Yaskawa INFORM job: vendrediTRJ4.JBI

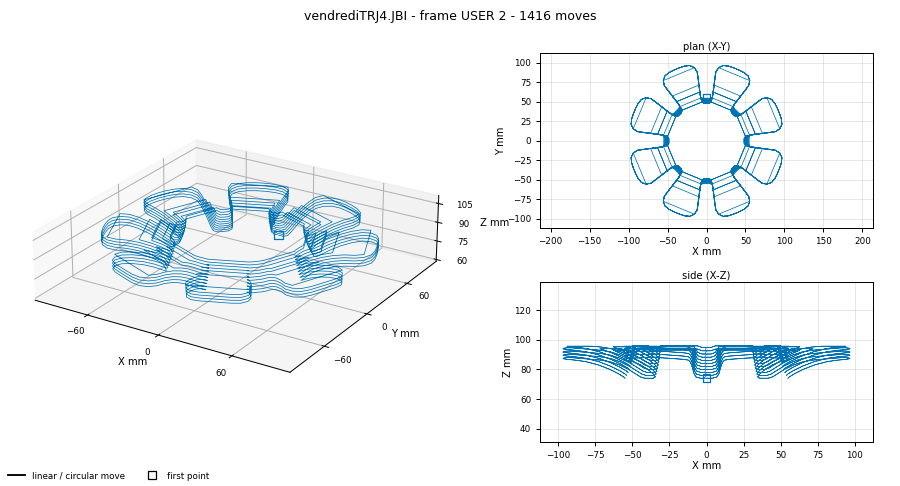
[picture p0: tool path of vendrediTRJ4.JBI in frame USER 2, 1416 of 1416 moves have a stored position in this frame; points joined in program order, loops and branches not executed]
/JOB
//NAME vendrediTRJ4
///FOLDERNAME DEMO
//POS
///NPOS 1416,0,1416,0,0,0
///USER 2
///TOOL 7
///POSTYPE USER
///RECTAN
///RCONF 1,0,0,0,0,0,0,0,0,0,0,0,0,0,0,0,0,0,0,0,0,0,0,0
C00000=0.000,54.840,74.049,-180.0000,29.7413,-14490.0000
C00001=1.666,54.823,74.024,-179.8067,29.7500,-14491.7406
C00002=4.048,54.790,74.062,173.8586,28.2915,-14494.2255
C00003=7.088,55.804,74.943,167.0788,9.5543,-14497.2387
C00004=8.393,59.388,77.145,-177.8370,-0.0706,-14498.0440
C00005=9.180,65.335,80.122,-176.4294,-0.0310,-14497.9981
C00006=10.089,72.980,83.074,-176.0907,-0.0153,-14497.8709
C00007=11.094,81.206,85.240,-175.9759,-0.0117,-14497.7793
C00008=12.226,88.613,86.276,-176.2817,-0.6456,-14497.8555
C00009=15.808,94.009,86.813,-178.2035,-1.5233,-14499.5452
C00010=21.475,96.642,87.246,-179.5823,-1.0342,-14502.5282
C00011=28.048,95.980,87.679,179.9973,-0.0724,-14506.2898
C00012=34.856,93.728,87.962,179.9966,-0.0074,-14510.3994
C00013=41.629,90.922,87.962,179.9972,-0.0076,-14514.6009
C00014=48.035,87.701,87.679,-179.9999,-0.0718,-14518.7101
C00015=53.151,83.521,87.246,179.5838,-1.0323,-14522.4718
C00016=55.296,77.652,86.813,178.2066,-1.5235,-14525.4547
C00017=54.014,71.304,86.276,176.2804,-0.6460,-14527.1446
C00018=49.577,65.266,85.240,175.9790,-0.0155,-14527.2208
C00019=44.470,58.738,83.074,176.0895,-0.0120,-14527.1290
C00020=39.708,52.690,80.122,176.4261,-0.0301,-14527.0022
C00021=36.059,47.928,77.145,177.8373,-0.0709,-14526.9563
C00022=34.447,44.472,74.943,-167.0757,9.5522,-14527.7605
C00023=35.880,41.605,74.062,-173.8568,28.2919,-14530.7744
C00024=37.588,39.944,74.024,179.8046,29.7498,-14533.2595
C00025=38.778,38.778,74.049,-180.0000,29.7416,-14535.0000
C00026=39.943,37.588,74.024,-179.8042,29.7498,-14536.7398
C00027=41.605,35.880,74.062,173.8533,28.2853,-14539.2256
C00028=44.472,34.447,74.943,167.0757,9.5522,-14542.2395
C00029=47.928,36.059,77.145,-177.8373,-0.0709,-14543.0437
C00030=52.690,39.708,80.122,-176.4261,-0.0301,-14542.9978
C00031=58.738,44.470,83.074,-176.0895,-0.0120,-14542.8710
C00032=65.266,49.577,85.240,-175.9790,-0.0155,-14542.7792
C00033=71.304,54.014,86.276,-176.2804,-0.6460,-14542.8554
C00034=77.652,55.296,86.813,-178.2066,-1.5235,-14544.5453
C00035=83.521,53.151,87.246,-179.5838,-1.0323,-14547.5282
C00036=87.701,48.035,87.679,179.9999,-0.0718,-14551.2899
C00037=90.922,41.629,87.962,-179.9972,-0.0076,-14555.3991
C00038=93.728,34.856,87.962,-179.9966,-0.0074,-14559.6006
C00039=95.980,28.048,87.679,-179.9973,-0.0724,-14563.7102
C00040=96.642,21.475,87.246,179.5823,-1.0342,-14567.4718
C00041=94.009,15.808,86.813,178.2035,-1.5233,-14570.4548
C00042=88.613,12.226,86.276,176.2817,-0.6456,-14572.1445
C00043=81.206,11.094,85.240,175.9759,-0.0117,-14572.2207
C00044=72.980,10.089,83.074,176.0907,-0.0153,-14572.1291
C00045=65.335,9.180,80.122,176.4294,-0.0310,-14572.0019
C00046=59.388,8.393,77.145,177.8370,-0.0706,-14571.9560
C00047=55.804,7.088,74.943,-167.0788,9.5543,-14572.7613
C00048=54.790,4.048,74.062,-173.8586,28.2915,-14575.7745
C00049=54.823,1.666,74.024,179.8067,29.7500,-14578.2594
C00050=54.840,0.000,74.049,180.0000,29.7413,-14580.0000
C00051=54.823,-1.665,74.024,-179.8061,29.7500,-14581.7396
C00052=54.790,-4.048,74.062,173.8593,28.2888,-14584.2255
C00053=55.804,-7.088,74.943,167.0788,9.5543,-14587.2387
C00054=59.388,-8.393,77.145,-177.8370,-0.0706,-14588.0440
C00055=65.335,-9.180,80.122,-176.4294,-0.0310,-14587.9981
C00056=72.980,-10.089,83.074,-176.0907,-0.0153,-14587.8709
C00057=81.206,-11.094,85.240,-175.9759,-0.0117,-14587.7793
C00058=88.613,-12.226,86.276,-176.2817,-0.6456,-14587.8555
C00059=94.009,-15.808,86.813,-178.2035,-1.5233,-14589.5452
C00060=96.642,-21.475,87.246,-179.5823,-1.0342,-14592.5282
C00061=95.980,-28.048,87.679,179.9973,-0.0724,-14596.2898
C00062=93.728,-34.856,87.962,179.9966,-0.0074,-14600.3994
C00063=90.922,-41.629,87.962,179.9972,-0.0076,-14604.6009
C00064=87.701,-48.035,87.679,-179.9999,-0.0718,-14608.7101
C00065=83.521,-53.151,87.246,179.5838,-1.0323,-14612.4718
C00066=77.652,-55.296,86.813,178.2066,-1.5235,-14615.4547
C00067=71.304,-54.014,86.276,176.2804,-0.6460,-14617.1446
C00068=65.266,-49.577,85.240,175.9790,-0.0155,-14617.2208
C00069=58.738,-44.470,83.074,176.0895,-0.0120,-14617.1290
C00070=52.690,-39.708,80.122,176.4261,-0.0301,-14617.0022
C00071=47.928,-36.059,77.145,177.8373,-0.0709,-14616.9563
C00072=44.472,-34.447,74.943,-167.0757,9.5522,-14617.7605
C00073=41.605,-35.880,74.062,-173.8568,28.2919,-14620.7744
C00074=39.944,-37.588,74.024,179.8046,29.7498,-14623.2595
C00075=38.778,-38.778,74.049,180.0000,29.7416,-14625.0000
C00076=37.588,-39.943,74.024,-179.8042,29.7498,-14626.7398
C00077=35.880,-41.605,74.062,173.8533,28.2853,-14629.2256
C00078=34.447,-44.472,74.943,167.0757,9.5522,-14632.2395
C00079=36.059,-47.928,77.145,-177.8373,-0.0709,-14633.0437
C00080=39.708,-52.690,80.122,-176.4261,-0.0301,-14632.9978
C00081=44.470,-58.738,83.074,-176.0895,-0.0120,-14632.8710
C00082=49.577,-65.266,85.240,-175.9790,-0.0155,-14632.7792
C00083=54.014,-71.304,86.276,-176.2804,-0.6460,-14632.8554
C00084=55.296,-77.652,86.813,-178.2066,-1.5235,-14634.5453
C00085=53.151,-83.521,87.246,-179.5838,-1.0323,-14637.5282
C00086=48.035,-87.701,87.679,179.9999,-0.0718,-14641.2899
C00087=41.629,-90.922,87.962,-179.9972,-0.0076,-14645.3991
C00088=34.856,-93.728,87.962,-179.9966,-0.0074,-14649.6006
C00089=28.048,-95.980,87.679,-179.9973,-0.0724,-14653.7102
C00090=21.475,-96.642,87.246,179.5823,-1.0342,-14657.4718
C00091=15.808,-94.009,86.813,178.2035,-1.5233,-14660.4548
C00092=12.226,-88.613,86.276,176.2817,-0.6456,-14662.1445
C00093=11.094,-81.206,85.240,175.9759,-0.0117,-14662.2207
C00094=10.089,-72.980,83.074,176.0907,-0.0153,-14662.1291
C00095=9.180,-65.335,80.122,176.4294,-0.0310,-14662.0019
C00096=8.393,-59.388,77.145,177.8370,-0.0706,-14661.9560
C00097=7.088,-55.804,74.943,-167.0788,9.5543,-14662.7613
C00098=4.048,-54.790,74.062,-173.8586,28.2915,-14665.7745
C00099=1.666,-54.823,74.024,179.8067,29.7500,-14668.2594
C00100=0.000,-54.840,74.049,-180.0000,29.7413,-14670.0000
C00101=-1.665,-54.823,74.024,-179.8061,29.7500,-14671.7396
C00102=-4.048,-54.790,74.062,173.8593,28.2888,-14674.2255
C00103=-7.088,-55.804,74.943,167.0788,9.5543,-14677.2387
C00104=-8.393,-59.388,77.145,-177.8370,-0.0706,-14678.0440
C00105=-9.180,-65.335,80.122,-176.4294,-0.0310,-14677.9981
C00106=-10.089,-72.980,83.074,-176.0907,-0.0153,-14677.8709
C00107=-11.094,-81.206,85.240,-175.9759,-0.0117,-14677.7793
C00108=-12.226,-88.613,86.276,-176.2817,-0.6456,-14677.8555
C00109=-15.808,-94.009,86.813,-178.2035,-1.5233,-14679.5452
C00110=-21.475,-96.642,87.246,-179.5823,-1.0342,-14682.5282
C00111=-28.048,-95.980,87.679,179.9973,-0.0724,-14686.2898
C00112=-34.856,-93.728,87.962,179.9966,-0.0074,-14690.3994
C00113=-41.629,-90.922,87.962,179.9972,-0.0076,-14694.6009
C00114=-48.035,-87.701,87.679,-179.9999,-0.0718,-14698.7101
C00115=-53.151,-83.521,87.246,179.5838,-1.0323,-14702.4718
C00116=-55.296,-77.652,86.813,178.2066,-1.5235,-14705.4547
C00117=-54.014,-71.304,86.276,176.2804,-0.6460,-14707.1446
C00118=-49.577,-65.266,85.240,175.9790,-0.0155,-14707.2208
C00119=-44.470,-58.738,83.074,176.0895,-0.0120,-14707.1290
C00120=-39.708,-52.690,80.122,176.4261,-0.0301,-14707.0022
C00121=-36.059,-47.928,77.145,177.8373,-0.0709,-14706.9563
C00122=-34.447,-44.472,74.943,-167.0757,9.5522,-14707.7605
C00123=-35.880,-41.605,74.062,-173.8568,28.2919,-14710.7744
C00124=-37.588,-39.944,74.024,179.8046,29.7498,-14713.2595
C00125=-38.778,-38.778,74.049,-180.0000,29.7416,-14715.0000
C00126=-39.943,-37.588,74.024,-179.8042,29.7498,-14716.7398
C00127=-41.605,-35.880,74.062,173.8533,28.2853,-14719.2256
C00128=-44.472,-34.447,74.943,167.0757,9.5522,-14722.2395
C00129=-47.928,-36.059,77.145,-177.8373,-0.0709,-14723.0437
C00130=-52.690,-39.708,80.122,-176.4261,-0.0301,-14722.9978
C00131=-58.738,-44.470,83.074,-176.0895,-0.0120,-14722.8710
C00132=-65.266,-49.577,85.240,-175.9790,-0.0155,-14722.7792
C00133=-71.304,-54.014,86.276,-176.2804,-0.6460,-14722.8554
C00134=-77.652,-55.296,86.813,-178.2066,-1.5235,-14724.5453
C00135=-83.521,-53.151,87.246,-179.5838,-1.0323,-14727.5282
C00136=-87.701,-48.035,87.679,179.9999,-0.0718,-14731.2899
C00137=-90.922,-41.629,87.962,-179.9972,-0.0076,-14735.3991
C00138=-93.728,-34.856,87.962,-179.9966,-0.0074,-14739.6006
C00139=-95.980,-28.048,87.679,-179.9973,-0.0724,-14743.7102
C00140=-96.642,-21.475,87.246,179.5823,-1.0342,-14747.4718
C00141=-94.009,-15.808,86.813,178.2035,-1.5233,-14750.4548
C00142=-88.613,-12.226,86.276,176.2817,-0.6456,-14752.1445
C00143=-81.206,-11.094,85.240,175.9759,-0.0117,-14752.2207
C00144=-72.980,-10.089,83.074,176.0907,-0.0153,-14752.1291
C00145=-65.335,-9.180,80.122,176.4294,-0.0310,-14752.0019
C00146=-59.388,-8.393,77.145,177.8370,-0.0706,-14751.9560
C00147=-55.804,-7.088,74.943,-167.0788,9.5543,-14752.7613
C00148=-54.790,-4.048,74.062,-173.8586,28.2915,-14755.7745
C00149=-54.823,-1.666,74.024,179.8067,29.7500,-14758.2594
C00150=-54.840,0.000,74.049,-180.0000,29.7413,-14760.0000
C00151=-54.823,1.665,74.024,-179.8061,29.7500,-14761.7396
C00152=-54.790,4.048,74.062,173.8593,28.2888,-14764.2255
C00153=-55.804,7.088,74.943,167.0788,9.5543,-14767.2387
C00154=-59.388,8.393,77.145,-177.8370,-0.0706,-14768.0440
C00155=-65.335,9.180,80.122,-176.4294,-0.0310,-14767.9981
C00156=-72.980,10.089,83.074,-176.0907,-0.0153,-14767.8709
C00157=-81.206,11.094,85.240,-175.9759,-0.0117,-14767.7793
C00158=-88.613,12.226,86.276,-176.2817,-0.6456,-14767.8555
C00159=-94.009,15.808,86.813,-178.2035,-1.5233,-14769.5452
C00160=-96.642,21.475,87.246,-179.5823,-1.0342,-14772.5282
C00161=-95.980,28.048,87.679,179.9973,-0.0724,-14776.2898
C00162=-93.728,34.856,87.962,179.9966,-0.0074,-14780.3994
C00163=-90.922,41.629,87.962,179.9972,-0.0076,-14784.6009
C00164=-87.701,48.035,87.679,-179.9999,-0.0718,-14788.7101
C00165=-83.521,53.151,87.246,179.5838,-1.0323,-14792.4718
C00166=-77.652,55.296,86.813,178.2066,-1.5235,-14795.4547
C00167=-71.304,54.014,86.276,176.2804,-0.6460,-14797.1446
C00168=-65.266,49.577,85.240,175.9790,-0.0155,-14797.2208
C00169=-58.738,44.470,83.074,176.0895,-0.0120,-14797.1290
C00170=-52.690,39.708,80.122,176.4261,-0.0301,-14797.0022
C00171=-47.928,36.059,77.145,177.8373,-0.0709,-14796.9563
C00172=-44.472,34.447,74.943,-167.0757,9.5522,-14797.7605
C00173=-41.605,35.880,74.062,-173.8568,28.2919,-14800.7744
C00174=-39.944,37.588,74.024,179.8046,29.7498,-14803.2595
C00175=-38.778,38.778,74.049,-180.0000,29.7416,-14805.0000
C00176=-37.588,39.943,74.024,-179.8042,29.7498,-14806.7398
C00177=-35.880,41.605,74.062,173.8533,28.2853,-14809.2256
C00178=-34.447,44.472,74.943,167.0757,9.5522,-14812.2395
C00179=-36.059,47.928,77.145,-177.8373,-0.0709,-14813.0437
C00180=-39.708,52.690,80.122,-176.4261,-0.0301,-14812.9978
C00181=-44.470,58.738,83.074,-176.0895,-0.0120,-14812.8710
C00182=-49.577,65.266,85.240,-175.9790,-0.0155,-14812.7792
C00183=-54.014,71.304,86.276,-176.2804,-0.6460,-14812.8554
C00184=-55.296,77.652,86.813,-178.2066,-1.5235,-14814.5453
C00185=-53.151,83.521,87.246,-179.5838,-1.0323,-14817.5282
C00186=-48.035,87.701,87.679,179.9999,-0.0718,-14821.2899
C00187=-41.629,90.922,87.962,-179.9972,-0.0076,-14825.3991
C00188=-34.856,93.728,87.962,-179.9966,-0.0074,-14829.6006
C00189=-28.048,95.980,87.679,-179.9973,-0.0724,-14833.7102
C00190=-21.475,96.642,87.246,179.5823,-1.0342,-14837.4718
C00191=-15.808,94.009,86.813,178.2035,-1.5233,-14840.4548
C00192=-12.226,88.613,86.276,176.2817,-0.6456,-14842.1445
C00193=-11.094,81.206,85.240,175.9759,-0.0117,-14842.2207
C00194=-10.089,72.980,83.074,176.0907,-0.0153,-14842.1291
C00195=-9.180,65.335,80.122,176.4294,-0.0310,-14842.0019
C00196=-8.393,59.388,77.145,177.8370,-0.0706,-14841.9560
C00197=-7.088,55.804,74.943,-167.0788,9.5543,-14842.7613
C00198=-4.048,54.790,74.062,-173.8593,28.2888,-14845.7745
C00199=-1.665,54.823,74.024,179.8061,29.7500,-14848.2604
C00200=0.000,53.776,75.975,180.0000,28.1001,-14850.0000
C00201=1.568,53.762,75.948,-179.8334,28.1117,-14851.6706
C00202=3.884,53.739,75.988,174.0567,26.6026,-14854.1339
C00203=6.894,54.818,76.900,168.1623,8.4382,-14857.1680
C00204=8.175,58.565,79.173,-177.8225,-0.0548,-14857.9465
C00205=8.965,64.737,82.228,-176.7507,-0.0188,-14857.8844
C00206=9.898,72.606,85.234,-176.6314,-0.0094,-14857.7630
C00207=10.924,81.005,87.424,-176.6961,-0.0057,-14857.6803
C00208=12.061,88.524,88.468,-177.0328,-0.5045,-14857.7585
C00209=15.662,93.991,89.008,-178.5867,-1.1939,-14859.4604
C00210=21.365,96.662,89.443,-179.6771,-0.7971,-14862.4636
C00211=27.983,96.002,89.878,179.9979,-0.0543,-14866.2505
C00212=34.834,93.736,90.162,-179.9980,-0.0054,-14870.3860
C00213=41.650,90.913,90.162,-179.9976,-0.0052,-14874.6140
C00214=48.097,87.670,89.878,179.9969,-0.0540,-14878.7498
C00215=53.243,83.458,89.443,179.6739,-0.7993,-14882.5363
C00216=55.387,77.537,89.008,178.5849,-1.1940,-14885.5394
C00217=54.067,71.124,88.468,177.0304,-0.5081,-14887.2413
C00218=49.554,65.004,87.424,176.6978,-0.0087,-14887.3191
C00219=44.341,58.339,85.234,176.6315,-0.0113,-14887.2369
C00220=39.437,52.115,82.228,176.7520,-0.0208,-14887.1159
C00221=35.631,47.192,79.173,177.8236,-0.0563,-14887.0536
C00222=33.888,43.637,76.900,-168.1624,8.4405,-14887.8325
C00223=35.253,40.746,75.988,-174.0559,26.5997,-14890.8660
C00224=36.906,39.124,75.948,179.8313,28.1098,-14893.3290
C00225=38.025,38.025,75.975,-180.0000,28.0967,-14895.0000
C00226=39.124,36.906,75.948,-179.8313,28.1098,-14896.6710
C00227=40.746,35.253,75.988,174.0559,26.5997,-14899.1340
C00228=43.637,33.888,76.901,168.1624,8.4405,-14902.1675
C00229=47.192,35.631,79.173,-177.8236,-0.0563,-14902.9464
C00230=52.115,39.437,82.228,-176.7520,-0.0208,-14902.8841
C00231=58.339,44.341,85.234,-176.6315,-0.0113,-14902.7631
C00232=65.004,49.554,87.424,-176.6978,-0.0087,-14902.6809
C00233=71.124,54.067,88.468,-177.0304,-0.5081,-14902.7587
C00234=77.537,55.387,89.008,-178.5849,-1.1940,-14904.4606
C00235=83.458,53.243,89.443,-179.6739,-0.7993,-14907.4637
C00236=87.670,48.097,89.878,-179.9969,-0.0540,-14911.2502
C00237=90.913,41.650,90.162,179.9976,-0.0052,-14915.3860
C00238=93.736,34.834,90.162,179.9980,-0.0054,-14919.6140
C00239=96.002,27.983,89.878,-179.9979,-0.0543,-14923.7495
C00240=96.662,21.365,89.443,179.6771,-0.7971,-14927.5364
C00241=93.991,15.662,89.008,178.5867,-1.1939,-14930.5396
C00242=88.524,12.061,88.468,177.0328,-0.5045,-14932.2415
C00243=81.005,10.924,87.424,176.6961,-0.0057,-14932.3197
C00244=72.606,9.898,85.234,176.6314,-0.0094,-14932.2370
C00245=64.737,8.965,82.228,176.7507,-0.0188,-14932.1156
C00246=58.565,8.175,79.173,177.8225,-0.0548,-14932.0535
C00247=54.818,6.894,76.900,-168.1623,8.4382,-14932.8320
C00248=53.739,3.884,75.988,-174.0567,26.6026,-14935.8661
C00249=53.762,1.568,75.948,179.8334,28.1117,-14938.3294
C00250=53.776,0.000,75.975,180.0000,28.1001,-14940.0000
C00251=53.762,-1.568,75.948,-179.8334,28.1117,-14941.6706
C00252=53.739,-3.885,75.988,174.0562,26.6025,-14944.1349
C00253=54.819,-6.894,76.901,168.1623,8.4383,-14947.1678
C00254=58.565,-8.175,79.173,-177.8225,-0.0548,-14947.9465
C00255=64.737,-8.965,82.228,-176.7507,-0.0188,-14947.8844
C00256=72.606,-9.898,85.234,-176.6314,-0.0094,-14947.7630
C00257=81.005,-10.924,87.424,-176.6961,-0.0057,-14947.6803
C00258=88.524,-12.061,88.468,-177.0328,-0.5045,-14947.7585
C00259=93.991,-15.662,89.008,-178.5867,-1.1939,-14949.4604
C00260=96.662,-21.365,89.443,-179.6771,-0.7971,-14952.4636
C00261=96.002,-27.983,89.878,179.9979,-0.0543,-14956.2505
C00262=93.736,-34.834,90.162,-179.9980,-0.0054,-14960.3860
C00263=90.913,-41.650,90.162,-179.9976,-0.0052,-14964.6140
C00264=87.670,-48.097,89.878,179.9969,-0.0540,-14968.7498
C00265=83.458,-53.243,89.443,179.6739,-0.7993,-14972.5363
C00266=77.537,-55.387,89.008,178.5849,-1.1940,-14975.5394
C00267=71.124,-54.067,88.468,177.0304,-0.5081,-14977.2413
C00268=65.004,-49.554,87.424,176.6978,-0.0087,-14977.3191
C00269=58.339,-44.341,85.234,176.6315,-0.0113,-14977.2369
C00270=52.115,-39.437,82.228,176.7520,-0.0208,-14977.1159
C00271=47.192,-35.631,79.173,177.8236,-0.0563,-14977.0536
C00272=43.637,-33.888,76.900,-168.1624,8.4405,-14977.8325
C00273=40.746,-35.253,75.988,-174.0559,26.5997,-14980.8660
C00274=39.124,-36.906,75.948,179.8313,28.1098,-14983.3290
C00275=38.025,-38.025,75.975,-180.0000,28.0967,-14985.0000
C00276=36.906,-39.124,75.948,-179.8313,28.1098,-14986.6710
C00277=35.253,-40.746,75.988,174.0559,26.5997,-14989.1340
C00278=33.888,-43.637,76.901,168.1624,8.4405,-14992.1675
C00279=35.631,-47.192,79.173,-177.8236,-0.0563,-14992.9464
C00280=39.437,-52.115,82.228,-176.7520,-0.0208,-14992.8841
C00281=44.341,-58.339,85.234,-176.6315,-0.0113,-14992.7631
C00282=49.554,-65.004,87.424,-176.6978,-0.0087,-14992.6809
C00283=54.067,-71.124,88.468,-177.0304,-0.5081,-14992.7587
C00284=55.387,-77.537,89.008,-178.5849,-1.1940,-14994.4606
C00285=53.243,-83.458,89.443,-179.6739,-0.7993,-14997.4637
C00286=48.097,-87.670,89.878,-179.9969,-0.0540,-15001.2502
C00287=41.650,-90.913,90.162,179.9976,-0.0052,-15005.3860
C00288=34.834,-93.736,90.162,179.9980,-0.0054,-15009.6140
C00289=27.983,-96.002,89.878,-179.9979,-0.0543,-15013.7495
C00290=21.365,-96.662,89.443,179.6771,-0.7971,-15017.5364
C00291=15.662,-93.991,89.008,178.5867,-1.1939,-15020.5396
C00292=12.061,-88.524,88.468,177.0328,-0.5045,-15022.2415
C00293=10.924,-81.005,87.424,176.6961,-0.0057,-15022.3197
C00294=9.898,-72.606,85.234,176.6314,-0.0094,-15022.2370
C00295=8.965,-64.737,82.228,176.7507,-0.0188,-15022.1156
C00296=8.175,-58.565,79.173,177.8225,-0.0548,-15022.0535
C00297=6.894,-54.818,76.900,-168.1623,8.4382,-15022.8320
C00298=3.884,-53.739,75.988,-174.0567,26.6026,-15025.8661
C00299=1.568,-53.762,75.948,179.8334,28.1117,-15028.3294
C00300=0.000,-53.776,75.975,180.0000,28.1001,-15030.0000
C00301=-1.568,-53.762,75.948,-179.8334,28.1117,-15031.6706
C00302=-3.885,-53.739,75.988,174.0562,26.6025,-15034.1349
C00303=-6.894,-54.819,76.901,168.1623,8.4383,-15037.1678
C00304=-8.175,-58.565,79.173,-177.8225,-0.0548,-15037.9465
C00305=-8.965,-64.737,82.228,-176.7507,-0.0188,-15037.8844
C00306=-9.898,-72.606,85.234,-176.6314,-0.0094,-15037.7630
C00307=-10.924,-81.005,87.424,-176.6961,-0.0057,-15037.6803
C00308=-12.061,-88.524,88.468,-177.0328,-0.5045,-15037.7585
C00309=-15.662,-93.991,89.008,-178.5867,-1.1939,-15039.4604
C00310=-21.365,-96.662,89.443,-179.6771,-0.7971,-15042.4636
C00311=-27.983,-96.002,89.878,179.9979,-0.0543,-15046.2505
C00312=-34.834,-93.736,90.162,-179.9980,-0.0054,-15050.3860
C00313=-41.650,-90.913,90.162,-179.9976,-0.0052,-15054.6140
C00314=-48.097,-87.670,89.878,179.9969,-0.0540,-15058.7498
C00315=-53.243,-83.458,89.443,179.6739,-0.7993,-15062.5363
C00316=-55.387,-77.537,89.008,178.5849,-1.1940,-15065.5394
C00317=-54.067,-71.124,88.468,177.0304,-0.5081,-15067.2413
C00318=-49.554,-65.004,87.424,176.6978,-0.0087,-15067.3191
C00319=-44.341,-58.339,85.234,176.6315,-0.0113,-15067.2369
C00320=-39.437,-52.115,82.228,176.7520,-0.0208,-15067.1159
C00321=-35.631,-47.192,79.173,177.8236,-0.0563,-15067.0536
C00322=-33.888,-43.637,76.900,-168.1624,8.4405,-15067.8325
C00323=-35.253,-40.746,75.988,-174.0559,26.5997,-15070.8660
C00324=-36.906,-39.124,75.948,179.8313,28.1098,-15073.3290
C00325=-38.025,-38.025,75.975,-180.0000,28.0967,-15075.0000
C00326=-39.124,-36.906,75.948,-179.8313,28.1098,-15076.6710
C00327=-40.746,-35.253,75.988,174.0559,26.5997,-15079.1340
C00328=-43.637,-33.888,76.901,168.1624,8.4405,-15082.1675
C00329=-47.192,-35.631,79.173,-177.8236,-0.0563,-15082.9464
C00330=-52.115,-39.437,82.228,-176.7520,-0.0208,-15082.8841
C00331=-58.339,-44.341,85.234,-176.6315,-0.0113,-15082.7631
C00332=-65.004,-49.554,87.424,-176.6978,-0.0087,-15082.6809
C00333=-71.124,-54.067,88.468,-177.0304,-0.5081,-15082.7587
C00334=-77.537,-55.387,89.008,-178.5849,-1.1940,-15084.4606
C00335=-83.458,-53.243,89.443,-179.6739,-0.7993,-15087.4637
C00336=-87.670,-48.097,89.878,-179.9969,-0.0540,-15091.2502
C00337=-90.913,-41.650,90.162,179.9976,-0.0052,-15095.3860
C00338=-93.736,-34.834,90.162,179.9980,-0.0054,-15099.6140
C00339=-96.002,-27.983,89.878,-179.9979,-0.0543,-15103.7495
C00340=-96.662,-21.365,89.443,179.6771,-0.7971,-15107.5364
C00341=-93.991,-15.662,89.008,178.5867,-1.1939,-15110.5396
C00342=-88.524,-12.061,88.468,177.0328,-0.5045,-15112.2415
C00343=-81.005,-10.924,87.424,176.6961,-0.0057,-15112.3197
C00344=-72.606,-9.898,85.234,176.6314,-0.0094,-15112.2370
C00345=-64.737,-8.965,82.228,176.7507,-0.0188,-15112.1156
C00346=-58.565,-8.175,79.173,177.8225,-0.0548,-15112.0535
C00347=-54.818,-6.894,76.900,-168.1623,8.4382,-15112.8320
C00348=-53.739,-3.884,75.988,-174.0567,26.6026,-15115.8661
C00349=-53.762,-1.568,75.948,179.8334,28.1117,-15118.3294
C00350=-53.776,0.000,75.975,180.0000,28.1001,-15120.0000
C00351=-53.762,1.568,75.948,-179.8334,28.1117,-15121.6706
C00352=-53.739,3.885,75.988,174.0562,26.6025,-15124.1349
C00353=-54.819,6.894,76.901,168.1623,8.4383,-15127.1678
C00354=-58.565,8.175,79.173,-177.8225,-0.0548,-15127.9465
C00355=-64.737,8.965,82.228,-176.7507,-0.0188,-15127.8844
C00356=-72.606,9.898,85.234,-176.6314,-0.0094,-15127.7630
C00357=-81.005,10.924,87.424,-176.6961,-0.0057,-15127.6803
C00358=-88.524,12.061,88.468,-177.0328,-0.5045,-15127.7585
C00359=-93.991,15.662,89.008,-178.5867,-1.1939,-15129.4604
C00360=-96.662,21.365,89.443,-179.6771,-0.7971,-15132.4636
C00361=-96.002,27.983,89.878,179.9979,-0.0543,-15136.2505
C00362=-93.736,34.834,90.162,-179.9980,-0.0054,-15140.3860
C00363=-90.913,41.650,90.162,-179.9976,-0.0052,-15144.6140
C00364=-87.670,48.097,89.878,179.9969,-0.0540,-15148.7498
C00365=-83.458,53.243,89.443,179.6739,-0.7993,-15152.5363
C00366=-77.537,55.387,89.008,178.5849,-1.1940,-15155.5394
C00367=-71.124,54.067,88.468,177.0304,-0.5081,-15157.2413
C00368=-65.004,49.554,87.424,176.6978,-0.0087,-15157.3191
C00369=-58.339,44.341,85.234,176.6315,-0.0113,-15157.2369
C00370=-52.115,39.437,82.228,176.7520,-0.0208,-15157.1159
C00371=-47.192,35.631,79.173,177.8236,-0.0563,-15157.0536
C00372=-43.637,33.888,76.900,-168.1624,8.4405,-15157.8325
C00373=-40.746,35.253,75.988,-174.0559,26.5997,-15160.8660
C00374=-39.124,36.906,75.948,179.8313,28.1098,-15163.3290
C00375=-38.025,38.025,75.975,-180.0000,28.0967,-15165.0000
C00376=-36.906,39.124,75.948,-179.8313,28.1098,-15166.6710
C00377=-35.253,40.746,75.988,174.0559,26.5997,-15169.1340
C00378=-33.888,43.637,76.901,168.1624,8.4405,-15172.1675
C00379=-35.631,47.192,79.173,-177.8236,-0.0563,-15172.9464
C00380=-39.437,52.115,82.228,-176.7520,-0.0208,-15172.8841
C00381=-44.341,58.339,85.234,-176.6315,-0.0113,-15172.7631
C00382=-49.554,65.004,87.424,-176.6978,-0.0087,-15172.6809
C00383=-54.067,71.124,88.468,-177.0304,-0.5081,-15172.7587
C00384=-55.387,77.537,89.008,-178.5849,-1.1940,-15174.4606
C00385=-53.243,83.458,89.443,-179.6739,-0.7993,-15177.4637
C00386=-48.097,87.670,89.878,-179.9969,-0.0540,-15181.2502
C00387=-41.650,90.913,90.162,179.9976,-0.0052,-15185.3860
C00388=-34.834,93.736,90.162,179.9980,-0.0054,-15189.6140
C00389=-27.983,96.002,89.878,-179.9979,-0.0543,-15193.7495
C00390=-21.365,96.662,89.443,179.6771,-0.7971,-15197.5364
C00391=-15.662,93.991,89.008,178.5867,-1.1939,-15200.5396
C00392=-12.061,88.524,88.468,177.0328,-0.5045,-15202.2415
C00393=-10.924,81.005,87.424,176.6961,-0.0057,-15202.3197
C00394=-9.898,72.606,85.234,176.6314,-0.0094,-15202.2370
C00395=-8.965,64.737,82.228,176.7507,-0.0188,-15202.1156
C00396=-8.175,58.565,79.173,177.8225,-0.0548,-15202.0535
C00397=-6.894,54.819,76.901,-168.1623,8.4383,-15202.8322
C00398=-3.885,53.739,75.988,-174.0562,26.6025,-15205.8651
C00399=-1.568,53.762,75.948,179.8334,28.1117,-15208.3294
C00400=0.000,52.771,77.932,-180.0000,26.2576,-15210.0000
C00401=1.476,52.759,77.904,-179.8644,26.2720,-15211.6025
C00402=3.730,52.747,77.945,174.3297,24.7331,-15214.0449
C00403=6.711,53.894,78.888,169.2924,7.3770,-15217.0981
C00404=7.974,57.808,81.229,-177.8824,-0.0435,-15217.8538
C00405=8.774,64.206,84.354,-177.1343,-0.0134,-15217.7815
C00406=9.737,72.291,87.405,-177.2235,-0.0020,-15217.6711
C00407=10.790,80.844,89.614,-177.4669,-0.0031,-15217.6022
C00408=11.935,88.455,90.663,-177.8347,-0.3615,-15217.6844
C00409=15.553,93.978,91.206,-179.0014,-0.8397,-15219.3971
C00410=21.285,96.677,91.642,-179.7804,-0.5442,-15222.4165
C00411=27.936,96.017,92.077,179.9986,-0.0362,-15226.2223
C00412=34.820,93.742,92.362,-179.9980,-0.0054,-15230.3773
C00413=41.664,90.907,92.362,-179.9976,-0.0052,-15234.6227
C00414=48.140,87.648,92.077,-179.9985,-0.0384,-15238.7775
C00415=53.310,83.412,91.642,179.7765,-0.5441,-15242.5833
C00416=55.455,77.451,91.206,179.0023,-0.8412,-15245.6027
C00417=54.108,70.986,90.663,177.8365,-0.3666,-15247.3159
C00418=49.536,64.795,89.614,177.4688,-0.0016,-15247.3980
C00419=44.233,58.003,87.405,177.2268,-0.0027,-15247.3291
C00420=39.197,51.604,84.354,177.1305,-0.0129,-15247.2193
C00421=35.238,46.514,81.229,177.8797,-0.0389,-15247.1468
C00422=33.363,42.854,78.888,-169.2963,7.3773,-15247.9017
C00423=34.660,39.935,77.945,-174.3268,24.7330,-15250.9551
C00424=36.262,38.350,77.904,179.8603,26.2704,-15253.3970
C00425=37.314,37.314,77.932,-180.0000,26.2558,-15255.0000
C00426=38.350,36.262,77.904,-179.8603,26.2704,-15256.6030
C00427=39.935,34.660,77.945,174.3268,24.7330,-15259.0449
C00428=42.854,33.363,78.888,169.2928,7.3727,-15262.0983
C00429=46.514,35.238,81.229,-177.8797,-0.0389,-15262.8532
C00430=51.604,39.197,84.354,-177.1305,-0.0129,-15262.7807
C00431=58.003,44.233,87.405,-177.2268,-0.0027,-15262.6709
C00432=64.795,49.536,89.614,-177.4688,-0.0016,-15262.6020
C00433=70.986,54.108,90.663,-177.8365,-0.3666,-15262.6841
C00434=77.451,55.455,91.206,-179.0023,-0.8412,-15264.3973
C00435=83.412,53.310,91.642,-179.7765,-0.5441,-15267.4167
C00436=87.648,48.140,92.077,179.9985,-0.0384,-15271.2225
C00437=90.907,41.664,92.362,179.9976,-0.0052,-15275.3773
C00438=93.742,34.820,92.362,179.9980,-0.0054,-15279.6227
C00439=96.017,27.936,92.077,-179.9986,-0.0362,-15283.7777
C00440=96.677,21.285,91.642,179.7804,-0.5442,-15287.5835
C00441=93.978,15.553,91.206,179.0014,-0.8397,-15290.6029
C00442=88.455,11.935,90.663,177.8347,-0.3615,-15292.3156
C00443=80.844,10.790,89.614,177.4669,-0.0031,-15292.3978
C00444=72.291,9.737,87.405,177.2235,-0.0020,-15292.3289
C00445=64.206,8.774,84.354,177.1343,-0.0134,-15292.2185
C00446=57.808,7.974,81.229,177.8824,-0.0435,-15292.1462
C00447=53.894,6.711,78.888,-169.2924,7.3770,-15292.9019
C00448=52.747,3.730,77.945,-174.3297,24.7331,-15295.9551
C00449=52.759,1.476,77.904,179.8644,26.2720,-15298.3975
C00450=52.771,0.000,77.932,-180.0000,26.2576,-15300.0000
C00451=52.759,-1.476,77.904,-179.8644,26.2720,-15301.6025
C00452=52.747,-3.730,77.945,174.3235,24.7327,-15304.0449
C00453=53.894,-6.711,78.888,169.2924,7.3770,-15307.0981
C00454=57.808,-7.974,81.229,-177.8824,-0.0435,-15307.8538
C00455=64.206,-8.774,84.354,-177.1343,-0.0134,-15307.7815
C00456=72.291,-9.737,87.405,-177.2235,-0.0020,-15307.6711
C00457=80.844,-10.790,89.614,-177.4669,-0.0031,-15307.6022
C00458=88.455,-11.935,90.663,-177.8347,-0.3615,-15307.6844
C00459=93.978,-15.553,91.206,-179.0014,-0.8397,-15309.3971
C00460=96.677,-21.285,91.642,-179.7804,-0.5442,-15312.4165
C00461=96.017,-27.936,92.077,179.9986,-0.0362,-15316.2223
C00462=93.742,-34.820,92.362,-179.9980,-0.0054,-15320.3773
C00463=90.907,-41.664,92.362,-179.9976,-0.0052,-15324.6227
C00464=87.648,-48.140,92.077,-179.9985,-0.0384,-15328.7775
C00465=83.412,-53.310,91.642,179.7765,-0.5441,-15332.5833
C00466=77.451,-55.455,91.206,179.0023,-0.8412,-15335.6027
C00467=70.986,-54.108,90.663,177.8365,-0.3666,-15337.3159
C00468=64.795,-49.536,89.614,177.4688,-0.0016,-15337.3980
C00469=58.003,-44.233,87.405,177.2268,-0.0027,-15337.3291
C00470=51.604,-39.197,84.354,177.1305,-0.0129,-15337.2193
C00471=46.514,-35.238,81.229,177.8797,-0.0389,-15337.1468
C00472=42.854,-33.363,78.888,-169.2963,7.3773,-15337.9017
C00473=39.935,-34.660,77.945,-174.3268,24.7330,-15340.9551
C00474=38.350,-36.262,77.904,179.8603,26.2704,-15343.3970
C00475=37.314,-37.314,77.932,180.0000,26.2558,-15345.0000
C00476=36.262,-38.350,77.904,-179.8603,26.2704,-15346.6030
C00477=34.660,-39.935,77.945,174.3268,24.7330,-15349.0449
C00478=33.363,-42.854,78.888,169.2928,7.3727,-15352.0983
C00479=35.238,-46.514,81.229,-177.8797,-0.0389,-15352.8532
C00480=39.197,-51.604,84.354,-177.1305,-0.0129,-15352.7807
C00481=44.233,-58.003,87.405,-177.2268,-0.0027,-15352.6709
C00482=49.536,-64.795,89.614,-177.4688,-0.0016,-15352.6020
C00483=54.108,-70.986,90.663,-177.8365,-0.3666,-15352.6841
C00484=55.455,-77.451,91.206,-179.0023,-0.8412,-15354.3973
C00485=53.310,-83.412,91.642,-179.7765,-0.5441,-15357.4167
C00486=48.140,-87.648,92.077,179.9985,-0.0384,-15361.2225
C00487=41.664,-90.907,92.362,179.9976,-0.0052,-15365.3773
C00488=34.820,-93.742,92.362,179.9980,-0.0054,-15369.6227
C00489=27.936,-96.017,92.077,-179.9986,-0.0362,-15373.7777
C00490=21.285,-96.677,91.642,179.7804,-0.5442,-15377.5835
C00491=15.553,-93.978,91.206,179.0014,-0.8397,-15380.6029
C00492=11.935,-88.455,90.663,177.8347,-0.3615,-15382.3156
C00493=10.790,-80.844,89.614,177.4669,-0.0031,-15382.3978
C00494=9.737,-72.291,87.405,177.2235,-0.0020,-15382.3289
C00495=8.774,-64.206,84.354,177.1343,-0.0134,-15382.2185
C00496=7.974,-57.808,81.229,177.8824,-0.0435,-15382.1462
C00497=6.711,-53.894,78.888,-169.2924,7.3770,-15382.9019
C00498=3.730,-52.747,77.945,-174.3297,24.7331,-15385.9551
C00499=1.476,-52.759,77.904,179.8644,26.2720,-15388.3975
C00500=0.000,-52.771,77.932,-180.0000,26.2576,-15390.0000
C00501=-1.476,-52.759,77.904,-179.8644,26.2720,-15391.6025
C00502=-3.730,-52.747,77.945,174.3235,24.7327,-15394.0449
C00503=-6.711,-53.894,78.888,169.2924,7.3770,-15397.0981
C00504=-7.974,-57.808,81.229,-177.8824,-0.0435,-15397.8538
C00505=-8.774,-64.206,84.354,-177.1343,-0.0134,-15397.7815
C00506=-9.737,-72.291,87.405,-177.2235,-0.0020,-15397.6711
C00507=-10.790,-80.844,89.614,-177.4669,-0.0031,-15397.6022
C00508=-11.935,-88.455,90.663,-177.8347,-0.3615,-15397.6844
C00509=-15.553,-93.978,91.206,-179.0014,-0.8397,-15399.3971
C00510=-21.285,-96.677,91.642,-179.7804,-0.5442,-15402.4165
C00511=-27.936,-96.017,92.077,179.9986,-0.0362,-15406.2223
C00512=-34.820,-93.742,92.362,-179.9980,-0.0054,-15410.3773
C00513=-41.664,-90.907,92.362,-179.9976,-0.0052,-15414.6227
C00514=-48.140,-87.648,92.077,-179.9985,-0.0384,-15418.7775
C00515=-53.310,-83.412,91.642,179.7765,-0.5441,-15422.5833
C00516=-55.455,-77.451,91.206,179.0023,-0.8412,-15425.6027
C00517=-54.108,-70.986,90.663,177.8365,-0.3666,-15427.3159
C00518=-49.536,-64.795,89.614,177.4688,-0.0016,-15427.3980
C00519=-44.233,-58.003,87.405,177.2268,-0.0027,-15427.3291
C00520=-39.197,-51.604,84.354,177.1305,-0.0129,-15427.2193
C00521=-35.238,-46.514,81.229,177.8797,-0.0389,-15427.1468
C00522=-33.363,-42.854,78.888,-169.2963,7.3773,-15427.9017
C00523=-34.660,-39.935,77.945,-174.3268,24.7330,-15430.9551
C00524=-36.262,-38.350,77.904,179.8603,26.2704,-15433.3970
C00525=-37.314,-37.314,77.932,180.0000,26.2558,-15435.0000
C00526=-38.350,-36.262,77.904,-179.8603,26.2704,-15436.6030
C00527=-39.935,-34.660,77.945,174.3268,24.7330,-15439.0449
C00528=-42.854,-33.363,78.888,169.2928,7.3727,-15442.0983
C00529=-46.514,-35.238,81.229,-177.8797,-0.0389,-15442.8532
C00530=-51.604,-39.197,84.354,-177.1305,-0.0129,-15442.7807
C00531=-58.003,-44.233,87.405,-177.2268,-0.0027,-15442.6709
C00532=-64.795,-49.536,89.614,-177.4688,-0.0016,-15442.6020
C00533=-70.986,-54.108,90.663,-177.8365,-0.3666,-15442.6841
C00534=-77.451,-55.455,91.206,-179.0023,-0.8412,-15444.3973
C00535=-83.412,-53.310,91.642,-179.7765,-0.5441,-15447.4167
C00536=-87.648,-48.140,92.077,179.9985,-0.0384,-15451.2225
C00537=-90.907,-41.664,92.362,179.9976,-0.0052,-15455.3773
C00538=-93.742,-34.820,92.362,179.9980,-0.0054,-15459.6227
C00539=-96.017,-27.936,92.077,-179.9986,-0.0362,-15463.7777
C00540=-96.677,-21.285,91.642,179.7804,-0.5442,-15467.5835
C00541=-93.978,-15.553,91.206,179.0014,-0.8397,-15470.6029
C00542=-88.455,-11.935,90.663,177.8347,-0.3615,-15472.3156
C00543=-80.844,-10.790,89.614,177.4669,-0.0031,-15472.3978
C00544=-72.291,-9.737,87.405,177.2235,-0.0020,-15472.3289
C00545=-64.206,-8.774,84.354,177.1343,-0.0134,-15472.2185
C00546=-57.808,-7.974,81.229,177.8824,-0.0435,-15472.1462
C00547=-53.894,-6.711,78.888,-169.2924,7.3770,-15472.9019
C00548=-52.747,-3.730,77.945,-174.3297,24.7331,-15475.9551
C00549=-52.759,-1.476,77.904,179.8644,26.2720,-15478.3975
C00550=-52.771,0.000,77.932,-180.0000,26.2576,-15480.0000
C00551=-52.759,1.476,77.904,-179.8644,26.2720,-15481.6025
C00552=-52.747,3.730,77.945,174.3235,24.7327,-15484.0449
C00553=-53.894,6.711,78.888,169.2924,7.3770,-15487.0981
C00554=-57.808,7.974,81.229,-177.8824,-0.0435,-15487.8538
C00555=-64.206,8.774,84.354,-177.1343,-0.0134,-15487.7815
C00556=-72.291,9.737,87.405,-177.2235,-0.0020,-15487.6711
C00557=-80.844,10.790,89.614,-177.4669,-0.0031,-15487.6022
C00558=-88.455,11.935,90.663,-177.8347,-0.3615,-15487.6844
C00559=-93.978,15.553,91.206,-179.0014,-0.8397,-15489.3971
C00560=-96.677,21.285,91.642,-179.7804,-0.5442,-15492.4165
C00561=-96.017,27.936,92.077,179.9986,-0.0362,-15496.2223
C00562=-93.742,34.820,92.362,-179.9980,-0.0054,-15500.3773
C00563=-90.907,41.664,92.362,-179.9976,-0.0052,-15504.6227
C00564=-87.648,48.140,92.077,-179.9985,-0.0384,-15508.7775
C00565=-83.412,53.310,91.642,179.7765,-0.5441,-15512.5833
C00566=-77.451,55.455,91.206,179.0023,-0.8412,-15515.6027
C00567=-70.986,54.108,90.663,177.8365,-0.3666,-15517.3159
C00568=-64.795,49.536,89.614,177.4688,-0.0016,-15517.3980
C00569=-58.003,44.233,87.405,177.2268,-0.0027,-15517.3291
C00570=-51.604,39.197,84.354,177.1305,-0.0129,-15517.2193
C00571=-46.514,35.238,81.229,177.8797,-0.0389,-15517.1468
C00572=-42.854,33.363,78.888,-169.2963,7.3773,-15517.9017
C00573=-39.935,34.660,77.945,-174.3268,24.7330,-15520.9551
C00574=-38.350,36.262,77.904,179.8603,26.2704,-15523.3970
C00575=-37.314,37.314,77.932,180.0000,26.2558,-15525.0000
C00576=-36.262,38.350,77.904,-179.8603,26.2704,-15526.6030
C00577=-34.660,39.935,77.945,174.3268,24.7330,-15529.0449
C00578=-33.363,42.854,78.888,169.2928,7.3727,-15532.0983
C00579=-35.238,46.514,81.229,-177.8797,-0.0389,-15532.8532
C00580=-39.197,51.604,84.354,-177.1305,-0.0129,-15532.7807
C00581=-44.233,58.003,87.405,-177.2268,-0.0027,-15532.6709
C00582=-49.536,64.795,89.614,-177.4688,-0.0016,-15532.6020
C00583=-54.108,70.986,90.663,-177.8365,-0.3666,-15532.6841
C00584=-55.455,77.451,91.206,-179.0023,-0.8412,-15534.3973
C00585=-53.310,83.412,91.642,-179.7765,-0.5441,-15537.4167
C00586=-48.140,87.648,92.077,179.9985,-0.0384,-15541.2225
C00587=-41.664,90.907,92.362,179.9976,-0.0052,-15545.3773
C00588=-34.820,93.742,92.362,179.9980,-0.0054,-15549.6227
C00589=-27.936,96.017,92.077,-179.9986,-0.0362,-15553.7777
C00590=-21.285,96.677,91.642,179.7804,-0.5442,-15557.5835
C00591=-15.553,93.978,91.206,179.0014,-0.8397,-15560.6029
C00592=-11.935,88.455,90.663,177.8347,-0.3615,-15562.3156
C00593=-10.790,80.844,89.614,177.4669,-0.0031,-15562.3978
C00594=-9.737,72.291,87.405,177.2235,-0.0020,-15562.3289
C00595=-8.774,64.206,84.354,177.1343,-0.0134,-15562.2185
C00596=-7.974,57.808,81.229,177.8824,-0.0435,-15562.1462
C00597=-6.711,53.894,78.888,-169.2924,7.3770,-15562.9019
C00598=-3.730,52.747,77.945,-174.3235,24.7327,-15565.9551
C00599=-1.476,52.759,77.904,179.8644,26.2720,-15568.3975
C00600=0.000,51.832,79.921,-180.0000,24.1993,-15570.0000
C00601=1.391,51.822,79.893,-179.8934,24.2117,-15571.5376
C00602=3.586,51.820,79.935,174.6728,22.6760,-15573.9586
C00603=6.543,53.038,80.908,170.4732,6.3608,-15577.0327
C00604=7.793,57.125,83.313,-178.0121,-0.0296,-15577.7683
C00605=8.610,63.749,86.500,-177.5700,-0.0072,-15577.6919
C00606=9.608,72.041,89.587,-177.8667,0.0012,-15577.5966
C00607=10.692,80.728,91.809,-178.2949,0.0004,-15577.5446
C00608=11.850,88.408,92.861,-178.6931,-0.2180,-15577.6343
C00609=15.484,93.970,93.405,-179.4470,-0.4664,-15579.3569
C00610=21.237,96.685,93.841,-179.8869,-0.2743,-15582.3884
C00611=27.910,96.026,94.277,179.9993,-0.0181,-15586.2065
C00612=34.811,93.745,94.562,-180.0000,-0.0000,-15590.3718
C00613=41.672,90.903,94.562,-180.0000,-0.0000,-15594.6278
C00614=48.166,87.636,94.277,-179.9995,-0.0128,-15598.7938
C00615=53.350,83.383,93.841,179.8851,-0.2776,-15602.6119
C00616=55.498,77.395,93.405,179.4467,-0.4673,-15605.6434
C00617=54.135,70.893,92.861,178.6953,-0.2176,-15607.3659
C00618=49.523,64.644,91.809,178.2957,0.0009,-15607.4553
C00619=44.146,57.735,89.587,177.8657,-0.0015,-15607.4027
C00620=38.990,51.166,86.500,177.5699,-0.0071,-15607.3085
C00621=34.883,45.903,83.313,178.0127,-0.0275,-15607.2322
C00622=32.877,42.130,80.908,-170.4687,6.3616,-15607.9674
C00623=34.107,39.178,79.935,-174.6789,22.6775,-15611.0417
C00624=35.661,37.627,79.893,179.8957,24.2122,-15613.4634
C00625=36.651,36.651,79.921,180.0000,24.1961,-15615.0000
C00626=37.627,35.661,79.893,-179.8914,24.2160,-15616.5366
C00627=39.178,34.107,79.935,174.6702,22.6769,-15618.9583
C00628=42.130,32.877,80.908,170.4687,6.3616,-15622.0326
C00629=45.903,34.883,83.313,-178.0127,-0.0275,-15622.7678
C00630=51.166,38.990,86.500,-177.5699,-0.0071,-15622.6915
C00631=57.735,44.146,89.587,-177.8657,-0.0015,-15622.5973
C00632=64.644,49.523,91.809,-178.2957,0.0009,-15622.5447
C00633=70.893,54.135,92.861,-178.6953,-0.2176,-15622.6341
C00634=77.395,55.498,93.405,-179.4467,-0.4673,-15624.3566
C00635=83.383,53.350,93.841,-179.8851,-0.2776,-15627.3881
C00636=87.636,48.166,94.277,179.9995,-0.0128,-15631.2062
C00637=90.903,41.672,94.562,-180.0000,-0.0000,-15635.3722
C00638=93.745,34.811,94.562,-180.0000,-0.0000,-15639.6282
C00639=96.026,27.910,94.277,-179.9993,-0.0181,-15643.7935
C00640=96.685,21.237,93.841,179.8869,-0.2743,-15647.6116
C00641=93.970,15.484,93.405,179.4470,-0.4664,-15650.6431
C00642=88.408,11.850,92.861,178.6931,-0.2180,-15652.3657
C00643=80.728,10.692,91.809,178.2949,0.0004,-15652.4554
C00644=72.041,9.608,89.587,177.8667,0.0012,-15652.4034
C00645=63.749,8.610,86.500,177.5700,-0.0072,-15652.3081
C00646=57.125,7.793,83.313,178.0121,-0.0296,-15652.2317
C00647=53.038,6.543,80.908,-170.4732,6.3608,-15652.9673
C00648=51.820,3.586,79.935,-174.6728,22.6760,-15656.0414
C00649=51.822,1.391,79.893,179.8934,24.2117,-15658.4624
C00650=51.832,0.000,79.921,-180.0000,24.1993,-15660.0000
C00651=51.822,-1.390,79.893,-179.8929,24.2117,-15661.5365
C00652=51.820,-3.586,79.935,174.6728,22.6760,-15663.9586
C00653=53.038,-6.543,80.908,170.4732,6.3608,-15667.0327
C00654=57.125,-7.793,83.313,-178.0121,-0.0296,-15667.7683
C00655=63.749,-8.610,86.500,-177.5700,-0.0072,-15667.6919
C00656=72.041,-9.608,89.587,-177.8667,0.0012,-15667.5966
C00657=80.728,-10.692,91.809,-178.2949,0.0004,-15667.5446
C00658=88.408,-11.850,92.861,-178.6931,-0.2180,-15667.6343
C00659=93.970,-15.484,93.405,-179.4470,-0.4664,-15669.3569
C00660=96.685,-21.237,93.841,-179.8869,-0.2743,-15672.3884
C00661=96.026,-27.910,94.277,179.9993,-0.0181,-15676.2065
C00662=93.745,-34.811,94.562,-180.0000,-0.0000,-15680.3718
C00663=90.903,-41.672,94.562,-180.0000,-0.0000,-15684.6278
C00664=87.636,-48.166,94.277,-179.9995,-0.0128,-15688.7938
C00665=83.383,-53.350,93.841,179.8851,-0.2776,-15692.6119
C00666=77.395,-55.498,93.405,179.4467,-0.4673,-15695.6434
C00667=70.893,-54.135,92.861,178.6953,-0.2176,-15697.3659
C00668=64.644,-49.523,91.809,178.2957,0.0009,-15697.4553
C00669=57.735,-44.146,89.587,177.8657,-0.0015,-15697.4027
C00670=51.166,-38.990,86.500,177.5699,-0.0071,-15697.3085
C00671=45.903,-34.883,83.313,178.0127,-0.0275,-15697.2322
C00672=42.130,-32.877,80.908,-170.4687,6.3616,-15697.9674
C00673=39.178,-34.107,79.935,-174.6789,22.6775,-15701.0417
C00674=37.627,-35.661,79.893,179.8957,24.2122,-15703.4634
C00675=36.651,-36.651,79.921,-180.0000,24.1961,-15705.0000
C00676=35.661,-37.627,79.893,-179.8914,24.2160,-15706.5366
C00677=34.107,-39.178,79.935,174.6702,22.6769,-15708.9583
C00678=32.877,-42.130,80.908,170.4687,6.3616,-15712.0326
C00679=34.883,-45.903,83.313,-178.0127,-0.0275,-15712.7678
C00680=38.990,-51.166,86.500,-177.5699,-0.0071,-15712.6915
C00681=44.146,-57.735,89.587,-177.8657,-0.0015,-15712.5973
C00682=49.523,-64.644,91.809,-178.2957,0.0009,-15712.5447
C00683=54.135,-70.893,92.861,-178.6953,-0.2176,-15712.6341
C00684=55.498,-77.395,93.405,-179.4467,-0.4673,-15714.3566
C00685=53.350,-83.383,93.841,-179.8851,-0.2776,-15717.3881
C00686=48.166,-87.636,94.277,179.9995,-0.0128,-15721.2062
C00687=41.672,-90.903,94.562,-180.0000,-0.0000,-15725.3722
C00688=34.811,-93.745,94.562,-180.0000,-0.0000,-15729.6282
C00689=27.910,-96.026,94.277,-179.9993,-0.0181,-15733.7935
C00690=21.237,-96.685,93.841,179.8869,-0.2743,-15737.6116
C00691=15.484,-93.970,93.405,179.4470,-0.4664,-15740.6431
C00692=11.850,-88.408,92.861,178.6931,-0.2180,-15742.3657
C00693=10.692,-80.728,91.809,178.2949,0.0004,-15742.4554
C00694=9.608,-72.041,89.587,177.8667,0.0012,-15742.4034
C00695=8.610,-63.749,86.500,177.5700,-0.0072,-15742.3081
C00696=7.793,-57.125,83.313,178.0121,-0.0296,-15742.2317
C00697=6.543,-53.038,80.908,-170.4732,6.3608,-15742.9673
C00698=3.586,-51.820,79.935,-174.6728,22.6760,-15746.0414
C00699=1.391,-51.822,79.893,179.8934,24.2117,-15748.4624
C00700=0.000,-51.832,79.921,180.0000,24.1993,-15750.0000
C00701=-1.390,-51.822,79.893,-179.8929,24.2117,-15751.5365
C00702=-3.586,-51.820,79.935,174.6728,22.6760,-15753.9586
C00703=-6.543,-53.038,80.908,170.4732,6.3608,-15757.0327
C00704=-7.793,-57.125,83.313,-178.0121,-0.0296,-15757.7683
C00705=-8.610,-63.749,86.500,-177.5700,-0.0072,-15757.6919
C00706=-9.608,-72.041,89.587,-177.8667,0.0012,-15757.5966
C00707=-10.692,-80.728,91.809,-178.2949,0.0004,-15757.5446
C00708=-11.850,-88.408,92.861,-178.6931,-0.2180,-15757.6343
C00709=-15.484,-93.970,93.405,-179.4470,-0.4664,-15759.3569
C00710=-21.237,-96.685,93.841,-179.8869,-0.2743,-15762.3884
C00711=-27.910,-96.026,94.277,179.9993,-0.0181,-15766.2065
C00712=-34.811,-93.745,94.562,-180.0000,-0.0000,-15770.3718
C00713=-41.672,-90.903,94.562,-180.0000,-0.0000,-15774.6278
C00714=-48.166,-87.636,94.277,-179.9995,-0.0128,-15778.7938
C00715=-53.350,-83.383,93.841,179.8851,-0.2776,-15782.6119
C00716=-55.498,-77.395,93.405,179.4467,-0.4673,-15785.6434
C00717=-54.135,-70.893,92.861,178.6953,-0.2176,-15787.3659
C00718=-49.523,-64.644,91.809,178.2957,0.0009,-15787.4553
C00719=-44.146,-57.735,89.587,177.8657,-0.0015,-15787.4027
C00720=-38.990,-51.166,86.500,177.5699,-0.0071,-15787.3085
C00721=-34.883,-45.903,83.313,178.0127,-0.0275,-15787.2322
C00722=-32.877,-42.130,80.908,-170.4687,6.3616,-15787.9674
C00723=-34.107,-39.178,79.935,-174.6789,22.6775,-15791.0417
C00724=-35.661,-37.627,79.893,179.8957,24.2122,-15793.4634
C00725=-36.651,-36.651,79.921,-180.0000,24.1961,-15795.0000
C00726=-37.627,-35.661,79.893,-179.8914,24.2160,-15796.5366
C00727=-39.178,-34.107,79.935,174.6702,22.6769,-15798.9583
C00728=-42.130,-32.877,80.908,170.4687,6.3616,-15802.0326
C00729=-45.903,-34.883,83.313,-178.0127,-0.0275,-15802.7678
C00730=-51.166,-38.990,86.500,-177.5699,-0.0071,-15802.6915
C00731=-57.735,-44.146,89.587,-177.8657,-0.0015,-15802.5973
C00732=-64.644,-49.523,91.809,-178.2957,0.0009,-15802.5447
C00733=-70.893,-54.135,92.861,-178.6953,-0.2176,-15802.6341
C00734=-77.395,-55.498,93.405,-179.4467,-0.4673,-15804.3566
C00735=-83.383,-53.350,93.841,-179.8851,-0.2776,-15807.3881
C00736=-87.636,-48.166,94.277,179.9995,-0.0128,-15811.2062
C00737=-90.903,-41.672,94.562,-180.0000,-0.0000,-15815.3722
C00738=-93.745,-34.811,94.562,-180.0000,-0.0000,-15819.6282
C00739=-96.026,-27.910,94.277,-179.9993,-0.0181,-15823.7935
C00740=-96.685,-21.237,93.841,179.8869,-0.2743,-15827.6116
C00741=-93.970,-15.484,93.405,179.4470,-0.4664,-15830.6431
C00742=-88.408,-11.850,92.861,178.6931,-0.2180,-15832.3657
C00743=-80.728,-10.692,91.809,178.2949,0.0004,-15832.4554
C00744=-72.041,-9.608,89.587,177.8667,0.0012,-15832.4034
C00745=-63.749,-8.610,86.500,177.5700,-0.0072,-15832.3081
C00746=-57.125,-7.793,83.313,178.0121,-0.0296,-15832.2317
C00747=-53.038,-6.543,80.908,-170.4732,6.3608,-15832.9673
C00748=-51.820,-3.586,79.935,-174.6728,22.6760,-15836.0414
C00749=-51.822,-1.391,79.893,179.8934,24.2117,-15838.4624
C00750=-51.832,0.000,79.921,180.0000,24.1993,-15840.0000
C00751=-51.822,1.390,79.893,-179.8929,24.2117,-15841.5365
C00752=-51.820,3.586,79.935,174.6728,22.6760,-15843.9586
C00753=-53.038,6.543,80.908,170.4732,6.3608,-15847.0327
C00754=-57.125,7.793,83.313,-178.0121,-0.0296,-15847.7683
C00755=-63.749,8.610,86.500,-177.5700,-0.0072,-15847.6919
C00756=-72.041,9.608,89.587,-177.8667,0.0012,-15847.5966
C00757=-80.728,10.692,91.809,-178.2949,0.0004,-15847.5446
C00758=-88.408,11.850,92.861,-178.6931,-0.2180,-15847.6343
C00759=-93.970,15.484,93.405,-179.4470,-0.4664,-15849.3569
C00760=-96.685,21.237,93.841,-179.8869,-0.2743,-15852.3884
C00761=-96.026,27.910,94.277,179.9993,-0.0181,-15856.2065
C00762=-93.745,34.811,94.562,-180.0000,-0.0000,-15860.3718
C00763=-90.903,41.672,94.562,-180.0000,-0.0000,-15864.6278
C00764=-87.636,48.166,94.277,-179.9995,-0.0128,-15868.7938
C00765=-83.383,53.350,93.841,179.8851,-0.2776,-15872.6119
C00766=-77.395,55.498,93.405,179.4467,-0.4673,-15875.6434
C00767=-70.893,54.135,92.861,178.6953,-0.2176,-15877.3659
C00768=-64.644,49.523,91.809,178.2957,0.0009,-15877.4553
C00769=-57.735,44.146,89.587,177.8657,-0.0015,-15877.4027
C00770=-51.166,38.990,86.500,177.5699,-0.0071,-15877.3085
C00771=-45.903,34.883,83.313,178.0127,-0.0275,-15877.2322
C00772=-42.130,32.877,80.908,-170.4687,6.3616,-15877.9674
C00773=-39.178,34.107,79.935,-174.6789,22.6775,-15881.0417
C00774=-37.627,35.661,79.893,179.8957,24.2122,-15883.4634
C00775=-36.651,36.651,79.921,-180.0000,24.1961,-15885.0000
C00776=-35.661,37.627,79.893,-179.8914,24.2160,-15886.5366
C00777=-34.107,39.178,79.935,174.6702,22.6769,-15888.9583
C00778=-32.877,42.130,80.908,170.4687,6.3616,-15892.0326
C00779=-34.883,45.903,83.313,-178.0127,-0.0275,-15892.7678
C00780=-38.990,51.166,86.500,-177.5699,-0.0071,-15892.6915
C00781=-44.146,57.735,89.587,-177.8657,-0.0015,-15892.5973
C00782=-49.523,64.644,91.809,-178.2957,0.0009,-15892.5447
C00783=-54.135,70.893,92.861,-178.6953,-0.2176,-15892.6341
C00784=-55.498,77.395,93.405,-179.4467,-0.4673,-15894.3566
C00785=-53.350,83.383,93.841,-179.8851,-0.2776,-15897.3881
C00786=-48.166,87.636,94.277,179.9995,-0.0128,-15901.2062
C00787=-41.672,90.903,94.562,-180.0000,-0.0000,-15905.3722
C00788=-34.811,93.745,94.562,-180.0000,-0.0000,-15909.6282
C00789=-27.910,96.026,94.277,-179.9993,-0.0181,-15913.7935
C00790=-21.237,96.685,93.841,179.8869,-0.2743,-15917.6116
C00791=-15.484,93.970,93.405,179.4470,-0.4664,-15920.6431
C00792=-11.850,88.408,92.861,178.6931,-0.2180,-15922.3657
C00793=-10.692,80.728,91.809,178.2949,0.0004,-15922.4554
C00794=-9.608,72.041,89.587,177.8667,0.0012,-15922.4034
C00795=-8.610,63.749,86.500,177.5700,-0.0072,-15922.3081
C00796=-7.793,57.125,83.313,178.0121,-0.0296,-15922.2317
C00797=-6.543,53.038,80.908,-170.4732,6.3608,-15922.9673
C00798=-3.586,51.820,79.935,-174.6728,22.6760,-15926.0414
C00799=-1.390,51.822,79.893,179.8929,24.2117,-15928.4635
C00800=0.000,50.970,81.946,180.0000,21.8993,-15930.0000
C00801=1.312,50.962,81.916,-179.9262,21.9171,-15931.4747
C00802=3.453,50.970,81.960,175.1064,20.4142,-15933.8756
C00803=6.389,52.261,82.960,171.6928,5.3944,-15936.9699
C00804=7.633,56.525,85.423,-178.2163,-0.0194,-15937.6906
C00805=8.475,63.374,88.663,-178.0565,-0.0061,-15937.6170
C00806=9.515,71.858,91.777,-178.5551,0.0006,-15937.5429
C00807=10.634,80.658,94.007,-179.1678,-0.0001,-15937.5106
C00808=11.808,88.386,95.061,-179.5979,-0.0677,-15937.6094
C00809=15.455,93.966,95.604,-179.9126,-0.0727,-15939.3401
C00810=55.516,77.372,95.604,179.9102,-0.0715,-15965.6602
C00811=54.149,70.847,95.061,179.5984,-0.0690,-15967.3910
C00812=49.515,64.553,94.007,179.1703,-0.0010,-15967.4898
C00813=44.083,57.539,91.777,178.5571,-0.0010,-15967.4572
C00814=38.820,50.805,88.663,178.0538,-0.0014,-15967.3834
C00815=34.571,45.367,85.423,178.2190,-0.0171,-15967.3085
C00816=32.436,41.472,82.960,-171.6874,5.3944,-15968.0296
C00817=33.599,38.483,81.960,-175.1072,20.4131,-15971.1238
C00818=35.108,36.963,81.916,179.9250,21.9192,-15973.5256
C00819=36.041,36.041,81.946,-180.0000,21.8955,-15975.0000
C00820=36.963,35.108,81.916,-179.9250,21.9192,-15976.4744
C00821=38.483,33.599,81.960,175.1072,20.4131,-15978.8762
C00822=41.472,32.436,82.960,171.6919,5.3909,-15981.9704
C00823=45.367,34.571,85.423,-178.2190,-0.0171,-15982.6915
C00824=50.805,38.820,88.663,-178.0538,-0.0014,-15982.6166
C00825=57.539,44.083,91.777,-178.5571,-0.0010,-15982.5428
C00826=64.553,49.515,94.007,-179.1703,-0.0010,-15982.5102
C00827=70.847,54.149,95.061,-179.5984,-0.0690,-15982.6090
C00828=77.372,55.516,95.604,-179.9102,-0.0715,-15984.3398
C00829=93.966,15.455,95.604,179.9126,-0.0727,-16010.6599
C00830=88.386,11.808,95.061,179.5979,-0.0677,-16012.3906
C00831=80.658,10.634,94.007,179.1678,-0.0001,-16012.4894
C00832=71.858,9.515,91.777,178.5551,0.0006,-16012.4571
C00833=63.374,8.475,88.663,178.0565,-0.0061,-16012.3830
C00834=56.525,7.633,85.423,178.2163,-0.0194,-16012.3094
C00835=52.261,6.389,82.960,-171.6928,5.3944,-16013.0301
C00836=50.970,3.453,81.960,-175.1064,20.4142,-16016.1244
C00837=50.962,1.312,81.916,179.9262,21.9171,-16018.5253
C00838=50.970,0.000,81.946,180.0000,21.8993,-16020.0000
C00839=50.962,-1.311,81.916,-179.9258,21.9171,-16021.4736
C00840=50.970,-3.454,81.960,175.1060,20.4141,-16023.8767
C00841=52.261,-6.389,82.960,171.6928,5.3944,-16026.9699
C00842=56.525,-7.633,85.423,-178.2163,-0.0194,-16027.6906
C00843=63.374,-8.475,88.663,-178.0565,-0.0061,-16027.6170
C00844=71.858,-9.515,91.777,-178.5551,0.0006,-16027.5429
C00845=80.658,-10.634,94.007,-179.1678,-0.0001,-16027.5106
C00846=88.386,-11.808,95.061,-179.5979,-0.0677,-16027.6094
C00847=93.966,-15.455,95.604,-179.9126,-0.0727,-16029.3401
C00848=77.372,-55.516,95.604,179.9102,-0.0715,-16055.6602
C00849=70.847,-54.149,95.061,179.5984,-0.0690,-16057.3910
C00850=64.553,-49.515,94.007,179.1703,-0.0010,-16057.4898
C00851=57.539,-44.083,91.777,178.5571,-0.0010,-16057.4572
C00852=50.805,-38.820,88.663,178.0538,-0.0014,-16057.3834
C00853=45.367,-34.571,85.423,178.2190,-0.0171,-16057.3085
C00854=41.472,-32.436,82.960,-171.6874,5.3944,-16058.0296
C00855=38.483,-33.599,81.960,-175.1072,20.4131,-16061.1238
C00856=36.963,-35.108,81.916,179.9250,21.9192,-16063.5256
C00857=36.041,-36.041,81.946,-180.0000,21.8955,-16065.0000
C00858=35.108,-36.963,81.916,-179.9250,21.9192,-16066.4744
C00859=33.599,-38.483,81.960,175.1072,20.4131,-16068.8762
C00860=32.436,-41.472,82.960,171.6919,5.3909,-16071.9704
C00861=34.571,-45.367,85.423,-178.2190,-0.0171,-16072.6915
C00862=38.820,-50.805,88.663,-178.0538,-0.0014,-16072.6166
C00863=44.083,-57.539,91.777,-178.5571,-0.0010,-16072.5428
C00864=49.515,-64.553,94.007,-179.1703,-0.0010,-16072.5102
C00865=54.149,-70.847,95.061,-179.5984,-0.0690,-16072.6090
C00866=55.516,-77.372,95.604,-179.9102,-0.0715,-16074.3398
C00867=15.455,-93.966,95.604,179.9126,-0.0727,-16100.6599
C00868=11.808,-88.386,95.061,179.5979,-0.0677,-16102.3906
C00869=10.634,-80.658,94.007,179.1678,-0.0001,-16102.4894
C00870=9.515,-71.858,91.777,178.5551,0.0006,-16102.4571
C00871=8.475,-63.374,88.663,178.0565,-0.0061,-16102.3830
C00872=7.633,-56.525,85.423,178.2163,-0.0194,-16102.3094
C00873=6.389,-52.261,82.960,-171.6928,5.3944,-16103.0301
C00874=3.453,-50.970,81.960,-175.1064,20.4142,-16106.1244
C00875=1.312,-50.962,81.916,179.9262,21.9171,-16108.5253
C00876=0.000,-50.970,81.946,180.0000,21.8993,-16110.0000
C00877=-1.311,-50.962,81.916,-179.9258,21.9171,-16111.4736
C00878=-3.454,-50.970,81.960,175.1060,20.4141,-16113.8767
C00879=-6.389,-52.261,82.960,171.6928,5.3944,-16116.9699
C00880=-7.633,-56.525,85.423,-178.2163,-0.0194,-16117.6906
C00881=-8.475,-63.374,88.663,-178.0565,-0.0061,-16117.6170
C00882=-9.515,-71.858,91.777,-178.5551,0.0006,-16117.5429
C00883=-10.634,-80.658,94.007,-179.1678,-0.0001,-16117.5106
C00884=-11.808,-88.386,95.061,-179.5979,-0.0677,-16117.6094
C00885=-15.455,-93.966,95.604,-179.9126,-0.0727,-16119.3401
C00886=-55.516,-77.372,95.604,179.9102,-0.0715,-16145.6602
C00887=-54.149,-70.847,95.061,179.5984,-0.0690,-16147.3910
C00888=-49.515,-64.553,94.007,179.1703,-0.0010,-16147.4898
C00889=-44.083,-57.539,91.777,178.5571,-0.0010,-16147.4572
C00890=-38.820,-50.805,88.663,178.0538,-0.0014,-16147.3834
C00891=-34.571,-45.367,85.423,178.2190,-0.0171,-16147.3085
C00892=-32.436,-41.472,82.960,-171.6874,5.3944,-16148.0296
C00893=-33.599,-38.483,81.960,-175.1072,20.4131,-16151.1238
C00894=-35.108,-36.963,81.916,179.9250,21.9192,-16153.5256
C00895=-36.041,-36.041,81.946,-180.0000,21.8955,-16155.0000
C00896=-36.963,-35.108,81.916,-179.9250,21.9192,-16156.4744
C00897=-38.483,-33.599,81.960,175.1072,20.4131,-16158.8762
C00898=-41.472,-32.436,82.960,171.6919,5.3909,-16161.9704
C00899=-45.367,-34.571,85.423,-178.2190,-0.0171,-16162.6915
C00900=-50.805,-38.820,88.663,-178.0538,-0.0014,-16162.6166
C00901=-57.539,-44.083,91.777,-178.5571,-0.0010,-16162.5428
C00902=-64.553,-49.515,94.007,-179.1703,-0.0010,-16162.5102
C00903=-70.847,-54.149,95.061,-179.5984,-0.0690,-16162.6090
C00904=-77.372,-55.516,95.604,-179.9102,-0.0715,-16164.3398
C00905=-93.966,-15.455,95.604,179.9126,-0.0727,-16190.6599
C00906=-88.386,-11.808,95.061,179.5979,-0.0677,-16192.3906
C00907=-80.658,-10.634,94.007,179.1678,-0.0001,-16192.4894
C00908=-71.858,-9.515,91.777,178.5551,0.0006,-16192.4571
C00909=-63.374,-8.475,88.663,178.0565,-0.0061,-16192.3830
C00910=-56.525,-7.633,85.423,178.2163,-0.0194,-16192.3094
C00911=-52.261,-6.389,82.960,-171.6928,5.3944,-16193.0301
C00912=-50.970,-3.453,81.960,-175.1064,20.4142,-16196.1244
C00913=-50.962,-1.312,81.916,179.9262,21.9171,-16198.5253
C00914=-50.970,0.000,81.946,-180.0000,21.8993,-16200.0000
C00915=-50.962,1.311,81.916,-179.9258,21.9171,-16201.4736
C00916=-50.970,3.454,81.960,175.1060,20.4141,-16203.8767
C00917=-52.261,6.389,82.960,171.6928,5.3944,-16206.9699
C00918=-56.525,7.633,85.423,-178.2163,-0.0194,-16207.6906
C00919=-63.374,8.475,88.663,-178.0565,-0.0061,-16207.6170
C00920=-71.858,9.515,91.777,-178.5551,0.0006,-16207.5429
C00921=-80.658,10.634,94.007,-179.1678,-0.0001,-16207.5106
C00922=-88.386,11.808,95.061,-179.5979,-0.0677,-16207.6094
C00923=-93.966,15.455,95.604,-179.9126,-0.0727,-16209.3401
C00924=-77.372,55.516,95.604,179.9102,-0.0715,-16235.6602
C00925=-70.847,54.149,95.061,179.5984,-0.0690,-16237.3910
C00926=-64.553,49.515,94.007,179.1703,-0.0010,-16237.4898
C00927=-57.539,44.083,91.777,178.5571,-0.0010,-16237.4572
C00928=-50.805,38.820,88.663,178.0538,-0.0014,-16237.3834
C00929=-45.367,34.571,85.423,178.2190,-0.0171,-16237.3085
C00930=-41.472,32.436,82.960,-171.6874,5.3944,-16238.0296
C00931=-38.483,33.599,81.960,-175.1072,20.4131,-16241.1238
C00932=-36.963,35.108,81.916,179.9250,21.9192,-16243.5256
C00933=-36.041,36.041,81.946,180.0000,21.8955,-16245.0000
C00934=-35.108,36.963,81.916,-179.9250,21.9192,-16246.4744
C00935=-33.599,38.483,81.960,175.1072,20.4131,-16248.8762
C00936=-32.436,41.472,82.960,171.6919,5.3909,-16251.9704
C00937=-34.571,45.367,85.423,-178.2190,-0.0171,-16252.6915
C00938=-38.820,50.805,88.663,-178.0538,-0.0014,-16252.6166
C00939=-44.083,57.539,91.777,-178.5571,-0.0010,-16252.5428
C00940=-49.515,64.553,94.007,-179.1703,-0.0010,-16252.5102
C00941=-54.149,70.847,95.061,-179.5984,-0.0690,-16252.6090
C00942=-55.516,77.372,95.604,-179.9102,-0.0715,-16254.3398
C00943=-15.455,93.966,95.604,179.9126,-0.0727,-16280.6599
C00944=-11.808,88.386,95.061,179.5979,-0.0677,-16282.3906
C00945=-10.634,80.658,94.007,179.1678,-0.0001,-16282.4894
C00946=-9.515,71.858,91.777,178.5551,0.0006,-16282.4571
C00947=-8.475,63.374,88.663,178.0565,-0.0061,-16282.3830
C00948=-7.633,56.525,85.423,178.2163,-0.0194,-16282.3094
C00949=-6.389,52.261,82.960,-171.6928,5.3944,-16283.0301
C00950=-3.454,50.970,81.960,-175.1060,20.4141,-16286.1233
C00951=-1.311,50.962,81.916,179.9258,21.9171,-16288.5264
C00952=0.000,50.195,84.004,-180.0000,19.3355,-16290.0000
C00953=1.241,50.188,83.974,-179.9511,19.3601,-16291.4165
C00954=3.334,50.204,84.019,175.6244,17.9316,-16293.7994
C00955=6.253,51.571,85.045,172.9492,4.4629,-16296.9134
C00956=7.499,56.017,87.559,-178.4839,-0.0109,-16297.6249
C00957=8.371,63.087,90.842,-178.5891,-0.0035,-16297.5584
C00958=9.459,71.748,93.974,-179.2893,0.0012,-16297.5104
C00959=44.045,57.421,93.974,179.2929,-0.0008,-16327.4901
C00960=38.690,50.529,90.842,178.5857,-0.0004,-16327.4412
C00961=34.307,44.912,87.559,178.4862,-0.0099,-16327.3752
C00962=32.045,40.888,85.045,-172.9480,4.4644,-16328.0867
C00963=33.142,37.857,84.019,-175.6236,17.9314,-16331.2006
C00964=34.611,36.365,83.974,179.9520,19.3612,-16333.5844
C00965=35.493,35.493,84.004,179.9957,19.3375,-16335.0000
C00966=36.365,34.611,83.974,-179.9520,19.3612,-16336.4156
C00967=37.858,33.142,84.019,175.6234,17.9313,-16338.8001
C00968=40.888,32.045,85.045,172.9480,4.4644,-16341.9133
C00969=44.912,34.307,87.559,-178.4862,-0.0099,-16342.6248
C00970=50.529,38.690,90.842,-178.5857,-0.0004,-16342.5588
C00971=57.421,44.045,93.974,-179.2929,-0.0008,-16342.5099
C00972=71.748,9.459,93.974,179.2893,0.0012,-16372.4896
C00973=63.087,8.371,90.842,178.5891,-0.0035,-16372.4416
C00974=56.017,7.499,87.559,178.4839,-0.0109,-16372.3751
C00975=51.571,6.253,85.045,-172.9492,4.4629,-16373.0866
C00976=50.204,3.334,84.019,-175.6244,17.9316,-16376.2006
C00977=50.188,1.241,83.974,179.9511,19.3601,-16378.5835
C00978=50.195,0.000,84.004,-180.0000,19.3355,-16380.0000
C00979=50.188,-1.240,83.974,-179.9507,19.3601,-16381.4153
C00980=50.204,-3.335,84.019,175.6241,17.9315,-16383.8005
C00981=51.571,-6.253,85.045,172.9492,4.4629,-16386.9134
C00982=56.017,-7.499,87.559,-178.4839,-0.0109,-16387.6249
C00983=63.087,-8.371,90.842,-178.5891,-0.0035,-16387.5584
C00984=71.748,-9.459,93.974,-179.2893,0.0012,-16387.5104
C00985=57.421,-44.045,93.974,179.2929,-0.0008,-16417.4901
C00986=50.529,-38.690,90.842,178.5857,-0.0004,-16417.4412
C00987=44.912,-34.307,87.559,178.4862,-0.0099,-16417.3752
C00988=40.888,-32.045,85.045,-172.9480,4.4644,-16418.0867
C00989=37.857,-33.142,84.019,-175.6236,17.9314,-16421.2006
C00990=36.365,-34.611,83.974,179.9520,19.3612,-16423.5844
C00991=35.493,-35.493,84.004,179.9957,19.3375,-16425.0000
C00992=34.611,-36.365,83.974,-179.9520,19.3612,-16426.4156
C00993=33.142,-37.858,84.019,175.6234,17.9313,-16428.8001
C00994=32.045,-40.888,85.045,172.9480,4.4644,-16431.9133
C00995=34.307,-44.912,87.559,-178.4862,-0.0099,-16432.6248
C00996=38.690,-50.529,90.842,-178.5857,-0.0004,-16432.5588
C00997=44.045,-57.421,93.974,-179.2929,-0.0008,-16432.5099
C00998=9.459,-71.748,93.974,179.2893,0.0012,-16462.4896
C00999=8.371,-63.087,90.842,178.5891,-0.0035,-16462.4416
C01000=7.499,-56.017,87.559,178.4839,-0.0109,-16462.3751
C01001=6.253,-51.571,85.045,-172.9492,4.4629,-16463.0866
C01002=3.334,-50.204,84.019,-175.6244,17.9316,-16466.2006
C01003=1.241,-50.188,83.974,179.9511,19.3601,-16468.5835
C01004=0.000,-50.195,84.004,-180.0000,19.3355,-16470.0000
C01005=-1.240,-50.188,83.974,-179.9507,19.3601,-16471.4153
C01006=-3.335,-50.204,84.019,175.6241,17.9315,-16473.8005
C01007=-6.253,-51.571,85.045,172.9492,4.4629,-16476.9134
C01008=-7.499,-56.017,87.559,-178.4839,-0.0109,-16477.6249
C01009=-8.371,-63.087,90.842,-178.5891,-0.0035,-16477.5584
C01010=-9.459,-71.748,93.974,-179.2893,0.0012,-16477.5104
C01011=-44.045,-57.421,93.974,179.2929,-0.0008,-16507.4901
C01012=-38.690,-50.529,90.842,178.5857,-0.0004,-16507.4412
C01013=-34.307,-44.912,87.559,178.4862,-0.0099,-16507.3752
C01014=-32.045,-40.888,85.045,-172.9480,4.4644,-16508.0867
C01015=-33.142,-37.857,84.019,-175.6236,17.9314,-16511.2006
C01016=-34.611,-36.365,83.974,179.9520,19.3612,-16513.5844
C01017=-35.493,-35.493,84.004,179.9957,19.3375,-16515.0000
C01018=-36.365,-34.611,83.974,-179.9520,19.3612,-16516.4156
C01019=-37.858,-33.142,84.019,175.6234,17.9313,-16518.8001
C01020=-40.888,-32.045,85.045,172.9480,4.4644,-16521.9133
C01021=-44.912,-34.307,87.559,-178.4862,-0.0099,-16522.6248
C01022=-50.529,-38.690,90.842,-178.5857,-0.0004,-16522.5588
C01023=-57.421,-44.045,93.974,-179.2929,-0.0008,-16522.5099
C01024=-71.748,-9.459,93.974,179.2893,0.0012,-16552.4896
C01025=-63.087,-8.371,90.842,178.5891,-0.0035,-16552.4416
C01026=-56.017,-7.499,87.559,178.4839,-0.0109,-16552.3751
C01027=-51.571,-6.253,85.045,-172.9492,4.4629,-16553.0866
C01028=-50.204,-3.334,84.019,-175.6244,17.9316,-16556.2006
C01029=-50.188,-1.241,83.974,179.9511,19.3601,-16558.5835
C01030=-50.195,0.000,84.004,-180.0000,19.3355,-16560.0000
C01031=-50.188,1.240,83.974,-179.9507,19.3601,-16561.4153
C01032=-50.204,3.335,84.019,175.6241,17.9315,-16563.8005
C01033=-51.571,6.253,85.045,172.9492,4.4629,-16566.9134
C01034=-56.017,7.499,87.559,-178.4839,-0.0109,-16567.6249
C01035=-63.087,8.371,90.842,-178.5891,-0.0035,-16567.5584
C01036=-71.748,9.459,93.974,-179.2893,0.0012,-16567.5104
C01037=-57.421,44.045,93.974,179.2929,-0.0008,-16597.4901
C01038=-50.529,38.690,90.842,178.5857,-0.0004,-16597.4412
C01039=-44.912,34.307,87.559,178.4862,-0.0099,-16597.3752
C01040=-40.888,32.045,85.045,-172.9480,4.4644,-16598.0867
C01041=-37.857,33.142,84.019,-175.6236,17.9314,-16601.2006
C01042=-36.365,34.611,83.974,179.9520,19.3612,-16603.5844
C01043=-35.493,35.493,84.004,179.9957,19.3375,-16605.0000
C01044=-34.611,36.365,83.974,-179.9520,19.3612,-16606.4156
C01045=-33.142,37.858,84.019,175.6234,17.9313,-16608.8001
C01046=-32.045,40.888,85.045,172.9480,4.4644,-16611.9133
C01047=-34.307,44.912,87.559,-178.4862,-0.0099,-16612.6248
C01048=-38.690,50.529,90.842,-178.5857,-0.0004,-16612.5588
C01049=-44.045,57.421,93.974,-179.2929,-0.0008,-16612.5099
C01050=-9.459,71.748,93.974,179.2893,0.0012,-16642.4896
C01051=-8.371,63.087,90.842,178.5891,-0.0035,-16642.4416
C01052=-7.499,56.017,87.559,178.4839,-0.0109,-16642.3751
C01053=-6.253,51.571,85.045,-172.9492,4.4629,-16643.0866
C01054=-3.335,50.204,84.019,-175.6241,17.9315,-16646.1995
C01055=-1.240,50.188,83.974,179.9507,19.3601,-16648.5847
C01056=0.000,49.517,86.097,-180.0000,16.4995,-16650.0000
C01057=1.179,49.510,86.067,-179.9745,16.5281,-16651.3641
C01058=3.230,49.536,86.112,176.2280,15.2268,-16653.7307
C01059=6.137,50.981,87.161,174.2492,3.5661,-16656.8641
C01060=7.391,55.610,89.719,-178.8088,-0.0035,-16657.5707
C01061=8.302,62.896,93.033,-179.1621,0.0008,-16657.5193
C01062=38.603,50.345,93.033,179.1623,0.0002,-16687.4799
C01063=34.096,44.548,89.719,178.8104,-0.0013,-16687.4296
C01064=31.710,40.389,87.161,-174.2479,3.5658,-16688.1360
C01065=32.743,37.311,86.112,-176.2272,15.2245,-16691.2692
C01066=34.176,35.843,86.067,179.9736,16.5280,-16693.6362
C01067=35.014,35.014,86.097,179.9958,16.5019,-16695.0000
C01068=35.842,34.176,86.067,-179.9734,16.5280,-16696.3630
C01069=37.311,32.743,86.112,176.2272,15.2245,-16698.7308
C01070=40.389,31.710,87.161,174.2524,3.5623,-16701.8640
C01071=44.548,34.096,89.719,-178.8104,-0.0013,-16702.5704
C01072=50.345,38.603,93.033,-179.1623,0.0002,-16702.5201
C01073=62.896,8.302,93.033,179.1621,0.0008,-16732.4807
C01074=55.610,7.391,89.719,178.8088,-0.0035,-16732.4293
C01075=50.981,6.137,87.161,-174.2492,3.5661,-16733.1359
C01076=49.536,3.230,86.112,-176.2280,15.2268,-16736.2693
C01077=49.510,1.179,86.067,179.9745,16.5281,-16738.6359
C01078=49.517,0.000,86.097,180.0000,16.4995,-16740.0000
C01079=49.510,-1.178,86.067,-179.9741,16.5281,-16741.3630
C01080=49.536,-3.231,86.112,176.2280,15.2212,-16743.7318
C01081=50.981,-6.137,87.161,174.2492,3.5661,-16746.8641
C01082=55.610,-7.391,89.719,-178.8088,-0.0035,-16747.5707
C01083=62.896,-8.302,93.033,-179.1621,0.0008,-16747.5193
C01084=50.345,-38.603,93.033,179.1623,0.0002,-16777.4799
C01085=44.548,-34.096,89.719,178.8104,-0.0013,-16777.4296
C01086=40.389,-31.710,87.161,-174.2479,3.5658,-16778.1360
C01087=37.311,-32.743,86.112,-176.2272,15.2245,-16781.2692
C01088=35.843,-34.176,86.067,179.9736,16.5280,-16783.6362
C01089=35.014,-35.014,86.097,179.9958,16.5019,-16785.0000
C01090=34.176,-35.842,86.067,-179.9734,16.5280,-16786.3630
C01091=32.743,-37.311,86.112,176.2272,15.2245,-16788.7308
C01092=31.710,-40.389,87.161,174.2524,3.5623,-16791.8640
C01093=34.096,-44.548,89.719,-178.8104,-0.0013,-16792.5704
C01094=38.603,-50.345,93.033,-179.1623,0.0002,-16792.5201
C01095=8.302,-62.896,93.033,179.1621,0.0008,-16822.4807
C01096=7.391,-55.610,89.719,178.8088,-0.0035,-16822.4293
C01097=6.137,-50.981,87.161,-174.2492,3.5661,-16823.1359
C01098=3.230,-49.536,86.112,-176.2280,15.2268,-16826.2693
C01099=1.179,-49.510,86.067,179.9745,16.5281,-16828.6359
C01100=0.000,-49.517,86.097,180.0000,16.4995,-16830.0000
C01101=-1.178,-49.510,86.067,-179.9741,16.5281,-16831.3630
C01102=-3.231,-49.536,86.112,176.2280,15.2212,-16833.7318
C01103=-6.137,-50.981,87.161,174.2492,3.5661,-16836.8641
C01104=-7.391,-55.610,89.719,-178.8088,-0.0035,-16837.5707
C01105=-8.302,-62.896,93.033,-179.1621,0.0008,-16837.5193
C01106=-38.603,-50.345,93.033,179.1623,0.0002,-16867.4799
C01107=-34.096,-44.548,89.719,178.8104,-0.0013,-16867.4296
C01108=-31.710,-40.389,87.161,-174.2479,3.5658,-16868.1360
C01109=-32.743,-37.311,86.112,-176.2272,15.2245,-16871.2692
C01110=-34.176,-35.843,86.067,179.9736,16.5280,-16873.6362
C01111=-35.014,-35.014,86.097,179.9958,16.5019,-16875.0000
C01112=-35.842,-34.176,86.067,-179.9734,16.5280,-16876.3630
C01113=-37.311,-32.743,86.112,176.2272,15.2245,-16878.7308
C01114=-40.389,-31.710,87.161,174.2524,3.5623,-16881.8640
C01115=-44.548,-34.096,89.719,-178.8104,-0.0013,-16882.5704
C01116=-50.345,-38.603,93.033,-179.1623,0.0002,-16882.5201
C01117=-62.896,-8.302,93.033,179.1621,0.0008,-16912.4807
C01118=-55.610,-7.391,89.719,178.8088,-0.0035,-16912.4293
C01119=-50.981,-6.137,87.161,-174.2492,3.5661,-16913.1359
C01120=-49.536,-3.230,86.112,-176.2280,15.2268,-16916.2693
C01121=-49.510,-1.179,86.067,179.9745,16.5281,-16918.6359
C01122=-49.517,0.000,86.097,180.0000,16.4995,-16920.0000
C01123=-49.510,1.178,86.067,-179.9741,16.5281,-16921.3630
C01124=-49.536,3.231,86.112,176.2280,15.2212,-16923.7318
C01125=-50.981,6.137,87.161,174.2492,3.5661,-16926.8641
C01126=-55.610,7.391,89.719,-178.8088,-0.0035,-16927.5707
C01127=-62.896,8.302,93.033,-179.1621,0.0008,-16927.5193
C01128=-50.345,38.603,93.033,179.1623,0.0002,-16957.4799
C01129=-44.548,34.096,89.719,178.8104,-0.0013,-16957.4296
C01130=-40.389,31.710,87.161,-174.2479,3.5658,-16958.1360
C01131=-37.311,32.743,86.112,-176.2272,15.2245,-16961.2692
C01132=-35.843,34.176,86.067,179.9736,16.5280,-16963.6362
C01133=-35.014,35.014,86.097,179.9958,16.5019,-16965.0000
C01134=-34.176,35.842,86.067,-179.9734,16.5280,-16966.3630
C01135=-32.743,37.311,86.112,176.2272,15.2245,-16968.7308
C01136=-31.710,40.389,87.161,174.2524,3.5623,-16971.8640
C01137=-34.096,44.548,89.719,-178.8104,-0.0013,-16972.5704
C01138=-38.603,50.345,93.033,-179.1623,0.0002,-16972.5201
C01139=-8.302,62.896,93.033,179.1621,0.0008,-17002.4807
C01140=-7.391,55.610,89.719,178.8088,-0.0035,-17002.4293
C01141=-6.137,50.981,87.161,-174.2492,3.5661,-17003.1359
C01142=-3.231,49.536,86.112,-176.2280,15.2212,-17006.2682
C01143=-1.178,49.510,86.067,179.9741,16.5281,-17008.6370
C01144=0.000,48.949,88.223,180.0000,13.3790,-17010.0000
C01145=1.127,48.942,88.191,-179.9906,13.4131,-17011.3191
C01146=3.143,48.975,88.238,176.9194,12.2840,-17013.6720
C01147=6.042,50.501,89.306,175.5912,2.6850,-17016.8225
C01148=7.312,55.314,91.898,-179.1905,-0.0028,-17017.5303
C01149=8.270,62.805,95.231,-179.7804,0.0000,-17017.5014
C01150=38.562,50.258,95.231,179.7754,0.0010,-17047.4983
C01151=33.942,44.284,91.898,179.1909,0.0007,-17047.4688
C01152=31.437,39.982,89.306,-175.5900,2.6894,-17048.1772
C01153=32.408,36.853,88.238,-176.9224,12.2833,-17051.3279
C01154=33.811,35.404,88.191,179.9936,13.4108,-17053.6816
C01155=34.612,34.612,88.223,-180.0000,13.3770,-17055.0000
C01156=35.404,33.811,88.191,-179.9936,13.4108,-17056.3184
C01157=36.854,32.408,88.238,176.9223,12.2833,-17058.6728
C01158=39.982,31.437,89.306,175.5945,2.6858,-17061.8228
C01159=44.284,33.942,91.898,-179.1909,0.0007,-17062.5312
C01160=50.258,38.562,95.231,-179.7754,0.0010,-17062.5017
C01161=62.805,8.270,95.231,179.7804,0.0000,-17092.4986
C01162=55.314,7.312,91.898,179.1905,-0.0028,-17092.4697
C01163=50.501,6.042,89.306,-175.5912,2.6850,-17093.1775
C01164=48.975,3.143,88.238,-176.9194,12.2840,-17096.3280
C01165=48.942,1.127,88.191,179.9906,13.4131,-17098.6809
C01166=48.949,0.000,88.223,-180.0000,13.3790,-17100.0000
C01167=48.942,-1.126,88.191,-179.9903,13.4131,-17101.3180
C01168=48.976,-3.143,88.238,176.9195,12.2840,-17103.6719
C01169=50.501,-6.042,89.306,175.5912,2.6850,-17106.8225
C01170=55.314,-7.312,91.898,-179.1905,-0.0028,-17107.5303
C01171=62.805,-8.270,95.231,-179.7804,0.0000,-17107.5014
C01172=50.258,-38.562,95.231,179.7754,0.0010,-17137.4983
C01173=44.284,-33.942,91.898,179.1909,0.0007,-17137.4688
C01174=39.982,-31.437,89.306,-175.5900,2.6894,-17138.1772
C01175=36.853,-32.408,88.238,-176.9224,12.2833,-17141.3279
C01176=35.404,-33.811,88.191,179.9936,13.4108,-17143.6816
C01177=34.612,-34.612,88.223,-180.0000,13.3770,-17145.0000
C01178=33.811,-35.404,88.191,-179.9936,13.4108,-17146.3184
C01179=32.408,-36.854,88.238,176.9223,12.2833,-17148.6728
C01180=31.437,-39.982,89.306,175.5945,2.6858,-17151.8228
C01181=33.942,-44.284,91.898,-179.1909,0.0007,-17152.5312
C01182=38.562,-50.258,95.231,-179.7754,0.0010,-17152.5017
C01183=8.270,-62.805,95.231,179.7804,0.0000,-17182.4986
C01184=7.312,-55.314,91.898,179.1905,-0.0028,-17182.4697
C01185=6.042,-50.501,89.306,-175.5912,2.6850,-17183.1775
C01186=3.143,-48.975,88.238,-176.9194,12.2840,-17186.3280
C01187=1.127,-48.942,88.191,179.9906,13.4131,-17188.6809
C01188=0.000,-48.949,88.223,-180.0000,13.3790,-17190.0000
C01189=-1.126,-48.942,88.191,-179.9903,13.4131,-17191.3180
C01190=-3.143,-48.976,88.238,176.9195,12.2840,-17193.6719
C01191=-6.042,-50.501,89.306,175.5912,2.6850,-17196.8225
C01192=-7.312,-55.314,91.898,-179.1905,-0.0028,-17197.5303
C01193=-8.270,-62.805,95.231,-179.7804,0.0000,-17197.5014
C01194=-38.562,-50.258,95.231,179.7754,0.0010,-17227.4983
C01195=-33.942,-44.284,91.898,179.1909,0.0007,-17227.4688
C01196=-31.437,-39.982,89.306,-175.5900,2.6894,-17228.1772
C01197=-32.408,-36.853,88.238,-176.9224,12.2833,-17231.3279
C01198=-33.811,-35.404,88.191,179.9936,13.4108,-17233.6816
C01199=-34.612,-34.612,88.223,180.0000,13.3770,-17235.0000
C01200=-35.404,-33.811,88.191,-179.9936,13.4108,-17236.3184
C01201=-36.854,-32.408,88.238,176.9223,12.2833,-17238.6728
C01202=-39.982,-31.437,89.306,175.5945,2.6858,-17241.8228
C01203=-44.284,-33.942,91.898,-179.1909,0.0007,-17242.5312
C01204=-50.258,-38.562,95.231,-179.7754,0.0010,-17242.5017
C01205=-62.805,-8.270,95.231,179.7804,0.0000,-17272.4986
C01206=-55.314,-7.312,91.898,179.1905,-0.0028,-17272.4697
C01207=-50.501,-6.042,89.306,-175.5912,2.6850,-17273.1775
C01208=-48.975,-3.143,88.238,-176.9194,12.2840,-17276.3280
C01209=-48.942,-1.127,88.191,179.9906,13.4131,-17278.6809
C01210=-48.949,0.000,88.223,-180.0000,13.3790,-17280.0000
C01211=-48.942,1.126,88.191,-179.9903,13.4131,-17281.3180
C01212=-48.976,3.143,88.238,176.9195,12.2840,-17283.6719
C01213=-50.501,6.042,89.306,175.5912,2.6850,-17286.8225
C01214=-55.314,7.312,91.898,-179.1905,-0.0028,-17287.5303
C01215=-62.805,8.270,95.231,-179.7804,0.0000,-17287.5014
C01216=-50.258,38.562,95.231,179.7754,0.0010,-17317.4983
C01217=-44.284,33.942,91.898,179.1909,0.0007,-17317.4688
C01218=-39.982,31.437,89.306,-175.5900,2.6894,-17318.1772
C01219=-36.853,32.408,88.238,-176.9224,12.2833,-17321.3279
C01220=-35.404,33.811,88.191,179.9936,13.4108,-17323.6816
C01221=-34.612,34.612,88.223,180.0000,13.3770,-17325.0000
C01222=-33.811,35.404,88.191,-179.9936,13.4108,-17326.3184
C01223=-32.408,36.854,88.238,176.9223,12.2833,-17328.6728
C01224=-31.437,39.982,89.306,175.5945,2.6858,-17331.8228
C01225=-33.942,44.284,91.898,-179.1909,0.0007,-17332.5312
C01226=-38.562,50.258,95.231,-179.7754,0.0010,-17332.5017
C01227=-8.270,62.805,95.231,179.7804,0.0000,-17362.4986
C01228=-7.312,55.314,91.898,179.1905,-0.0028,-17362.4697
C01229=-6.042,50.501,89.306,-175.5912,2.6850,-17363.1775
C01230=-3.143,48.976,88.238,-176.9195,12.2840,-17366.3281
C01231=-1.126,48.942,88.191,179.9903,13.4131,-17368.6820
C01232=0.000,48.503,90.377,-180.0000,9.9625,-17370.0000
C01233=1.086,48.496,90.345,-179.9994,10.0055,-17371.2828
C01234=3.075,48.536,90.393,177.6967,9.1102,-17373.6251
C01235=5.972,50.143,91.476,176.9766,1.8184,-17376.7919
C01236=7.266,55.138,94.090,-179.6070,-0.0002,-17377.5071
C01237=33.851,44.126,94.090,179.6115,-0.0019,-17407.4934
C01238=31.234,39.679,91.476,-176.9779,1.8180,-17408.2087
C01239=32.146,36.494,90.393,-177.6994,9.1088,-17411.3754
C01240=33.524,35.059,90.345,-179.9960,10.0034,-17413.7178
C01241=34.297,34.297,90.377,180.0000,9.9681,-17415.0000
C01242=35.059,33.525,90.345,179.9962,10.0034,-17416.2813
C01243=36.495,32.146,90.393,177.6954,9.1045,-17418.6253
C01244=39.679,31.234,91.476,176.9779,1.8180,-17421.7913
C01245=44.126,33.851,94.090,-179.6115,-0.0019,-17422.5066
C01246=55.138,7.266,94.090,179.6070,-0.0002,-17452.4929
C01247=50.143,5.972,91.476,-176.9766,1.8184,-17453.2081
C01248=48.536,3.075,90.393,-177.6967,9.1102,-17456.3749
C01249=48.496,1.086,90.345,179.9994,10.0055,-17458.7172
C01250=48.503,0.000,90.377,-180.0000,9.9625,-17460.0000
C01251=48.496,-1.085,90.345,-179.9992,10.0055,-17461.2817
C01252=48.536,-3.075,90.393,177.6967,9.1102,-17463.6251
C01253=50.143,-5.972,91.476,176.9766,1.8184,-17466.7919
C01254=55.138,-7.266,94.090,-179.6070,-0.0002,-17467.5071
C01255=44.126,-33.851,94.090,179.6115,-0.0019,-17497.4934
C01256=39.679,-31.234,91.476,-176.9779,1.8180,-17498.2087
C01257=36.494,-32.146,90.393,-177.6994,9.1088,-17501.3754
C01258=35.059,-33.524,90.345,-179.9960,10.0034,-17503.7178
C01259=34.297,-34.297,90.377,180.0000,9.9681,-17505.0000
C01260=33.525,-35.059,90.345,179.9962,10.0034,-17506.2813
C01261=32.146,-36.495,90.393,177.6954,9.1045,-17508.6253
C01262=31.234,-39.679,91.476,176.9779,1.8180,-17511.7913
C01263=33.851,-44.126,94.090,-179.6115,-0.0019,-17512.5066
C01264=7.266,-55.138,94.090,179.6070,-0.0002,-17542.4929
C01265=5.972,-50.143,91.476,-176.9766,1.8184,-17543.2081
C01266=3.075,-48.536,90.393,-177.6967,9.1102,-17546.3749
C01267=1.086,-48.496,90.345,179.9994,10.0055,-17548.7172
C01268=0.000,-48.503,90.377,-180.0000,9.9625,-17550.0000
C01269=-1.085,-48.496,90.345,-179.9992,10.0055,-17551.2817
C01270=-3.075,-48.536,90.393,177.6967,9.1102,-17553.6251
C01271=-5.972,-50.143,91.476,176.9766,1.8184,-17556.7919
C01272=-7.266,-55.138,94.090,-179.6070,-0.0002,-17557.5071
C01273=-33.851,-44.126,94.090,179.6115,-0.0019,-17587.4934
C01274=-31.234,-39.679,91.476,-176.9779,1.8180,-17588.2087
C01275=-32.146,-36.494,90.393,-177.6994,9.1088,-17591.3754
C01276=-33.524,-35.059,90.345,-179.9960,10.0034,-17593.7178
C01277=-34.297,-34.297,90.377,-180.0000,9.9681,-17595.0000
C01278=-35.059,-33.525,90.345,179.9962,10.0034,-17596.2813
C01279=-36.495,-32.146,90.393,177.6954,9.1045,-17598.6253
C01280=-39.679,-31.234,91.476,176.9779,1.8180,-17601.7913
C01281=-44.126,-33.851,94.090,-179.6115,-0.0019,-17602.5066
C01282=-55.138,-7.266,94.090,179.6070,-0.0002,-17632.4929
C01283=-50.143,-5.972,91.476,-176.9766,1.8184,-17633.2081
C01284=-48.536,-3.075,90.393,-177.6967,9.1102,-17636.3749
C01285=-48.496,-1.086,90.345,179.9994,10.0055,-17638.7172
C01286=-48.503,0.000,90.377,-180.0000,9.9625,-17640.0000
C01287=-48.496,1.085,90.345,-179.9992,10.0055,-17641.2817
C01288=-48.536,3.075,90.393,177.6967,9.1102,-17643.6251
C01289=-50.143,5.972,91.476,176.9766,1.8184,-17646.7919
C01290=-55.138,7.266,94.090,-179.6070,-0.0002,-17647.5071
C01291=-44.126,33.851,94.090,179.6115,-0.0019,-17677.4934
C01292=-39.679,31.234,91.476,-176.9779,1.8180,-17678.2087
C01293=-36.494,32.146,90.393,-177.6994,9.1088,-17681.3754
C01294=-35.059,33.524,90.345,-179.9960,10.0034,-17683.7178
C01295=-34.297,34.297,90.377,-180.0000,9.9681,-17685.0000
C01296=-33.525,35.059,90.345,179.9962,10.0034,-17686.2813
C01297=-32.146,36.495,90.393,177.6954,9.1045,-17688.6253
C01298=-31.234,39.679,91.476,176.9779,1.8180,-17691.7913
C01299=-33.851,44.126,94.090,-179.6115,-0.0019,-17692.5066
C01300=-7.266,55.138,94.090,179.6070,-0.0002,-17722.4929
C01301=-5.972,50.143,91.476,-176.9766,1.8184,-17723.2081
C01302=-3.075,48.536,90.393,-177.6967,9.1102,-17726.3749
C01303=-1.085,48.496,90.345,179.9992,10.0055,-17728.7183
C01304=0.000,48.191,92.555,180.0000,6.2750,-17730.0000
C01305=1.057,48.183,92.523,179.9934,6.3226,-17731.2567
C01306=3.027,48.229,92.571,178.5501,5.7076,-17733.5913
C01307=5.927,49.917,93.664,178.4157,0.9490,-17736.7714
C01308=31.106,39.488,93.664,-178.4140,0.9504,-17768.2287
C01309=31.963,36.244,92.571,-178.5471,5.7094,-17771.4086
C01310=33.323,34.818,92.523,-179.9953,6.3224,-17773.7431
C01311=34.076,34.076,92.555,-180.0000,6.2761,-17775.0000
C01312=34.818,33.324,92.523,179.9954,6.3224,-17776.2560
C01313=36.244,31.963,92.571,178.5471,5.7094,-17778.5914
C01314=39.488,31.106,93.664,178.4140,0.9504,-17781.7713
C01315=49.917,5.927,93.664,-178.4157,0.9490,-17813.2286
C01316=48.229,3.027,92.571,-178.5501,5.7076,-17816.4087
C01317=48.183,1.057,92.523,-179.9934,6.3226,-17818.7433
C01318=48.191,0.000,92.555,180.0000,6.2750,-17820.0000
C01319=48.183,-1.057,92.523,179.9934,6.3226,-17821.2567
C01320=48.229,-3.027,92.571,178.5443,5.7073,-17823.5913
C01321=49.918,-5.927,93.664,178.4157,0.9490,-17826.7713
C01322=39.488,-31.106,93.664,-178.4140,0.9504,-17858.2287
C01323=36.244,-31.963,92.571,-178.5471,5.7094,-17861.4086
C01324=34.818,-33.323,92.523,-179.9953,6.3224,-17863.7431
C01325=34.076,-34.076,92.555,-180.0000,6.2761,-17865.0000
C01326=33.324,-34.818,92.523,179.9954,6.3224,-17866.2560
C01327=31.963,-36.244,92.571,178.5471,5.7094,-17868.5914
C01328=31.106,-39.488,93.664,178.4140,0.9504,-17871.7713
C01329=5.927,-49.917,93.664,-178.4157,0.9490,-17903.2286
C01330=3.027,-48.229,92.571,-178.5501,5.7076,-17906.4087
C01331=1.057,-48.183,92.523,-179.9934,6.3226,-17908.7433
C01332=0.000,-48.191,92.555,180.0000,6.2750,-17910.0000
C01333=-1.057,-48.183,92.523,179.9934,6.3226,-17911.2567
C01334=-3.027,-48.229,92.571,178.5443,5.7073,-17913.5913
C01335=-5.927,-49.918,93.664,178.4157,0.9490,-17916.7713
C01336=-31.106,-39.488,93.664,-178.4140,0.9504,-17948.2287
C01337=-31.963,-36.244,92.571,-178.5471,5.7094,-17951.4086
C01338=-33.323,-34.818,92.523,-179.9953,6.3224,-17953.7431
C01339=-34.076,-34.076,92.555,-180.0000,6.2761,-17955.0000
C01340=-34.818,-33.324,92.523,179.9954,6.3224,-17956.2560
C01341=-36.244,-31.963,92.571,178.5471,5.7094,-17958.5914
C01342=-39.488,-31.106,93.664,178.4140,0.9504,-17961.7713
C01343=-49.917,-5.927,93.664,-178.4157,0.9490,-17993.2286
C01344=-48.229,-3.027,92.571,-178.5501,5.7076,-17996.4087
C01345=-48.183,-1.057,92.523,-179.9934,6.3226,-17998.7433
C01346=-48.191,0.000,92.555,180.0000,6.2750,-18000.0000
C01347=-48.183,1.057,92.523,179.9934,6.3226,-18001.2567
C01348=-48.229,3.027,92.571,178.5443,5.7073,-18003.5913
C01349=-49.918,5.927,93.664,178.4157,0.9490,-18006.7713
C01350=-39.488,31.106,93.664,-178.4140,0.9504,-18038.2287
C01351=-36.244,31.963,92.571,-178.5471,5.7094,-18041.4086
C01352=-34.818,33.323,92.523,-179.9953,6.3224,-18043.7431
C01353=-34.076,34.076,92.555,-180.0000,6.2761,-18045.0000
C01354=-33.324,34.818,92.523,179.9954,6.3224,-18046.2560
C01355=-31.963,36.244,92.571,178.5471,5.7094,-18048.5914
C01356=-31.106,39.488,93.664,178.4140,0.9504,-18051.7713
C01357=-5.927,49.918,93.664,-178.4157,0.9490,-18083.2287
C01358=-3.027,48.229,92.571,-178.5443,5.7073,-18086.4087
C01359=-1.057,48.183,92.523,-179.9934,6.3226,-18088.7433
C01360=0.000,48.026,94.749,-180.0000,2.3325,-18090.0000
C01361=1.042,48.016,94.716,179.9997,2.3906,-18091.2432
C01362=3.002,48.067,94.764,179.4608,2.1024,-18093.5737
C01363=5.911,49.834,95.862,179.9066,0.0582,-18096.7645
C01364=31.058,39.418,95.862,-179.9039,0.0539,-18128.2351
C01365=31.866,36.111,94.764,-179.4625,2.1022,-18131.4267
C01366=33.216,34.689,94.716,-179.9968,2.3916,-18133.7573
C01367=33.959,33.959,94.749,180.0000,2.3342,-18135.0000
C01368=34.689,33.216,94.716,179.9968,2.3916,-18136.2427
C01369=36.111,31.865,94.764,179.4624,2.1022,-18138.5742
C01370=39.418,31.058,95.862,179.9039,0.0539,-18141.7649
C01371=49.834,5.911,95.862,-179.9066,0.0582,-18173.2355
C01372=48.067,3.002,94.764,-179.4608,2.1024,-18176.4263
C01373=48.016,1.042,94.716,-179.9997,2.3906,-18178.7568
C01374=48.026,0.000,94.749,-180.0000,2.3325,-18180.0000
C01375=48.016,-1.041,94.716,179.9998,2.3906,-18181.2420
C01376=48.067,-3.002,94.764,179.4608,2.1024,-18183.5737
C01377=49.834,-5.911,95.862,179.9066,0.0582,-18186.7645
C01378=39.418,-31.058,95.862,-179.9039,0.0539,-18218.2351
C01379=36.111,-31.866,94.764,-179.4625,2.1022,-18221.4267
C01380=34.689,-33.216,94.716,-179.9968,2.3916,-18223.7573
C01381=33.959,-33.959,94.749,180.0000,2.3342,-18225.0000
C01382=33.216,-34.689,94.716,179.9968,2.3916,-18226.2427
C01383=31.865,-36.111,94.764,179.4624,2.1022,-18228.5742
C01384=31.058,-39.418,95.862,179.9039,0.0539,-18231.7649
C01385=5.911,-49.834,95.862,-179.9066,0.0582,-18263.2355
C01386=3.002,-48.067,94.764,-179.4608,2.1024,-18266.4263
C01387=1.042,-48.016,94.716,-179.9997,2.3906,-18268.7568
C01388=0.000,-48.026,94.749,-180.0000,2.3325,-18270.0000
C01389=-1.041,-48.016,94.716,179.9998,2.3906,-18271.2420
C01390=-3.002,-48.067,94.764,179.4608,2.1024,-18273.5737
C01391=-5.911,-49.834,95.862,179.9066,0.0582,-18276.7645
C01392=-31.058,-39.418,95.862,-179.9039,0.0539,-18308.2351
C01393=-31.866,-36.111,94.764,-179.4625,2.1022,-18311.4267
C01394=-33.216,-34.689,94.716,-179.9968,2.3916,-18313.7573
C01395=-33.959,-33.959,94.749,180.0000,2.3342,-18315.0000
C01396=-34.689,-33.216,94.716,179.9968,2.3916,-18316.2427
C01397=-36.111,-31.865,94.764,179.4624,2.1022,-18318.5742
C01398=-39.418,-31.058,95.862,179.9039,0.0539,-18321.7649
C01399=-49.834,-5.911,95.862,-179.9066,0.0582,-18353.2355
C01400=-48.067,-3.002,94.764,-179.4608,2.1024,-18356.4263
C01401=-48.016,-1.042,94.716,-179.9997,2.3906,-18358.7568
C01402=-48.026,0.000,94.749,-180.0000,2.3325,-18360.0000
C01403=-48.016,1.041,94.716,179.9998,2.3906,-18361.2420
C01404=-48.067,3.002,94.764,179.4608,2.1024,-18363.5737
C01405=-49.834,5.911,95.862,179.9066,0.0582,-18366.7645
C01406=-39.418,31.058,95.862,-179.9039,0.0539,-18398.2351
C01407=-36.111,31.866,94.764,-179.4625,2.1022,-18401.4267
C01408=-34.689,33.216,94.716,-179.9968,2.3916,-18403.7573
C01409=-33.959,33.959,94.749,180.0000,2.3342,-18405.0000
C01410=-33.216,34.689,94.716,179.9968,2.3916,-18406.2427
C01411=-31.865,36.111,94.764,179.4624,2.1022,-18408.5742
C01412=-31.058,39.418,95.862,179.9039,0.0539,-18411.7649
C01413=-5.911,49.834,95.862,-179.9066,0.0582,-18443.2355
C01414=-3.002,48.067,94.764,-179.4608,2.1024,-18446.4263
C01415=-1.041,48.016,94.716,-179.9998,2.3906,-18448.7580
///TOOL 0
///POSTYPE ANGLE
///ANGLE
EC00000=29.7413,14490.0000
EC00001=29.7500,14491.7406
EC00002=28.2915,14494.2255
EC00003=9.5543,14497.2387
EC00004=-0.0706,14498.0440
EC00005=-0.0310,14497.9981
EC00006=-0.0153,14497.8709
EC00007=-0.0117,14497.7793
EC00008=-0.6456,14497.8555
EC00009=-1.5233,14499.5452
EC00010=-1.0342,14502.5282
EC00011=-0.0724,14506.2898
EC00012=-0.0074,14510.3994
EC00013=-0.0076,14514.6009
EC00014=-0.0718,14518.7101
EC00015=-1.0323,14522.4718
EC00016=-1.5235,14525.4547
EC00017=-0.6460,14527.1446
EC00018=-0.0155,14527.2208
EC00019=-0.0120,14527.1290
EC00020=-0.0301,14527.0022
EC00021=-0.0709,14526.9563
EC00022=9.5522,14527.7605
EC00023=28.2919,14530.7744
EC00024=29.7498,14533.2595
EC00025=29.7416,14535.0000
EC00026=29.7498,14536.7398
EC00027=28.2853,14539.2256
EC00028=9.5522,14542.2395
EC00029=-0.0709,14543.0437
EC00030=-0.0301,14542.9978
EC00031=-0.0120,14542.8710
EC00032=-0.0155,14542.7792
EC00033=-0.6460,14542.8554
EC00034=-1.5235,14544.5453
EC00035=-1.0323,14547.5282
EC00036=-0.0718,14551.2899
EC00037=-0.0076,14555.3991
EC00038=-0.0074,14559.6006
EC00039=-0.0724,14563.7102
EC00040=-1.0342,14567.4718
EC00041=-1.5233,14570.4548
EC00042=-0.6456,14572.1445
EC00043=-0.0117,14572.2207
EC00044=-0.0153,14572.1291
EC00045=-0.0310,14572.0019
EC00046=-0.0706,14571.9560
EC00047=9.5543,14572.7613
EC00048=28.2915,14575.7745
EC00049=29.7500,14578.2594
EC00050=29.7413,14580.0000
EC00051=29.7500,14581.7396
EC00052=28.2888,14584.2255
EC00053=9.5543,14587.2387
EC00054=-0.0706,14588.0440
EC00055=-0.0310,14587.9981
EC00056=-0.0153,14587.8709
EC00057=-0.0117,14587.7793
EC00058=-0.6456,14587.8555
EC00059=-1.5233,14589.5452
EC00060=-1.0342,14592.5282
EC00061=-0.0724,14596.2898
EC00062=-0.0074,14600.3994
EC00063=-0.0076,14604.6009
EC00064=-0.0718,14608.7101
EC00065=-1.0323,14612.4718
EC00066=-1.5235,14615.4547
EC00067=-0.6460,14617.1446
EC00068=-0.0155,14617.2208
EC00069=-0.0120,14617.1290
EC00070=-0.0301,14617.0022
EC00071=-0.0709,14616.9563
EC00072=9.5522,14617.7605
EC00073=28.2919,14620.7744
EC00074=29.7498,14623.2595
EC00075=29.7416,14625.0000
EC00076=29.7498,14626.7398
EC00077=28.2853,14629.2256
EC00078=9.5522,14632.2395
EC00079=-0.0709,14633.0437
EC00080=-0.0301,14632.9978
EC00081=-0.0120,14632.8710
EC00082=-0.0155,14632.7792
EC00083=-0.6460,14632.8554
EC00084=-1.5235,14634.5453
EC00085=-1.0323,14637.5282
EC00086=-0.0718,14641.2899
EC00087=-0.0076,14645.3991
EC00088=-0.0074,14649.6006
EC00089=-0.0724,14653.7102
EC00090=-1.0342,14657.4718
EC00091=-1.5233,14660.4548
EC00092=-0.6456,14662.1445
EC00093=-0.0117,14662.2207
EC00094=-0.0153,14662.1291
EC00095=-0.0310,14662.0019
EC00096=-0.0706,14661.9560
EC00097=9.5543,14662.7613
EC00098=28.2915,14665.7745
EC00099=29.7500,14668.2594
EC00100=29.7413,14670.0000
EC00101=29.7500,14671.7396
EC00102=28.2888,14674.2255
EC00103=9.5543,14677.2387
EC00104=-0.0706,14678.0440
EC00105=-0.0310,14677.9981
EC00106=-0.0153,14677.8709
EC00107=-0.0117,14677.7793
EC00108=-0.6456,14677.8555
EC00109=-1.5233,14679.5452
EC00110=-1.0342,14682.5282
EC00111=-0.0724,14686.2898
EC00112=-0.0074,14690.3994
EC00113=-0.0076,14694.6009
EC00114=-0.0718,14698.7101
EC00115=-1.0323,14702.4718
EC00116=-1.5235,14705.4547
EC00117=-0.6460,14707.1446
EC00118=-0.0155,14707.2208
EC00119=-0.0120,14707.1290
EC00120=-0.0301,14707.0022
EC00121=-0.0709,14706.9563
EC00122=9.5522,14707.7605
EC00123=28.2919,14710.7744
EC00124=29.7498,14713.2595
EC00125=29.7416,14715.0000
EC00126=29.7498,14716.7398
EC00127=28.2853,14719.2256
EC00128=9.5522,14722.2395
EC00129=-0.0709,14723.0437
EC00130=-0.0301,14722.9978
EC00131=-0.0120,14722.8710
EC00132=-0.0155,14722.7792
EC00133=-0.6460,14722.8554
EC00134=-1.5235,14724.5453
EC00135=-1.0323,14727.5282
EC00136=-0.0718,14731.2899
EC00137=-0.0076,14735.3991
EC00138=-0.0074,14739.6006
EC00139=-0.0724,14743.7102
EC00140=-1.0342,14747.4718
EC00141=-1.5233,14750.4548
EC00142=-0.6456,14752.1445
EC00143=-0.0117,14752.2207
EC00144=-0.0153,14752.1291
EC00145=-0.0310,14752.0019
EC00146=-0.0706,14751.9560
EC00147=9.5543,14752.7613
EC00148=28.2915,14755.7745
EC00149=29.7500,14758.2594
EC00150=29.7413,14760.0000
EC00151=29.7500,14761.7396
EC00152=28.2888,14764.2255
EC00153=9.5543,14767.2387
EC00154=-0.0706,14768.0440
EC00155=-0.0310,14767.9981
EC00156=-0.0153,14767.8709
EC00157=-0.0117,14767.7793
EC00158=-0.6456,14767.8555
EC00159=-1.5233,14769.5452
EC00160=-1.0342,14772.5282
EC00161=-0.0724,14776.2898
EC00162=-0.0074,14780.3994
EC00163=-0.0076,14784.6009
EC00164=-0.0718,14788.7101
EC00165=-1.0323,14792.4718
EC00166=-1.5235,14795.4547
EC00167=-0.6460,14797.1446
EC00168=-0.0155,14797.2208
EC00169=-0.0120,14797.1290
EC00170=-0.0301,14797.0022
EC00171=-0.0709,14796.9563
EC00172=9.5522,14797.7605
EC00173=28.2919,14800.7744
EC00174=29.7498,14803.2595
EC00175=29.7416,14805.0000
EC00176=29.7498,14806.7398
EC00177=28.2853,14809.2256
EC00178=9.5522,14812.2395
EC00179=-0.0709,14813.0437
EC00180=-0.0301,14812.9978
EC00181=-0.0120,14812.8710
EC00182=-0.0155,14812.7792
EC00183=-0.6460,14812.8554
EC00184=-1.5235,14814.5453
EC00185=-1.0323,14817.5282
EC00186=-0.0718,14821.2899
EC00187=-0.0076,14825.3991
EC00188=-0.0074,14829.6006
EC00189=-0.0724,14833.7102
EC00190=-1.0342,14837.4718
EC00191=-1.5233,14840.4548
EC00192=-0.6456,14842.1445
EC00193=-0.0117,14842.2207
EC00194=-0.0153,14842.1291
EC00195=-0.0310,14842.0019
EC00196=-0.0706,14841.9560
EC00197=9.5543,14842.7613
EC00198=28.2888,14845.7745
EC00199=29.7500,14848.2604
EC00200=28.1001,14850.0000
EC00201=28.1117,14851.6706
EC00202=26.6026,14854.1339
EC00203=8.4382,14857.1680
EC00204=-0.0548,14857.9465
EC00205=-0.0188,14857.8844
EC00206=-0.0094,14857.7630
EC00207=-0.0057,14857.6803
EC00208=-0.5045,14857.7585
EC00209=-1.1939,14859.4604
EC00210=-0.7971,14862.4636
EC00211=-0.0543,14866.2505
EC00212=-0.0054,14870.3860
EC00213=-0.0052,14874.6140
EC00214=-0.0540,14878.7498
EC00215=-0.7993,14882.5363
EC00216=-1.1940,14885.5394
EC00217=-0.5081,14887.2413
EC00218=-0.0087,14887.3191
EC00219=-0.0113,14887.2369
EC00220=-0.0208,14887.1159
EC00221=-0.0563,14887.0536
EC00222=8.4405,14887.8325
EC00223=26.5997,14890.8660
EC00224=28.1098,14893.3290
EC00225=28.0967,14895.0000
EC00226=28.1098,14896.6710
EC00227=26.5997,14899.1340
EC00228=8.4405,14902.1675
EC00229=-0.0563,14902.9464
EC00230=-0.0208,14902.8841
EC00231=-0.0113,14902.7631
EC00232=-0.0087,14902.6809
EC00233=-0.5081,14902.7587
EC00234=-1.1940,14904.4606
EC00235=-0.7993,14907.4637
EC00236=-0.0540,14911.2502
EC00237=-0.0052,14915.3860
EC00238=-0.0054,14919.6140
EC00239=-0.0543,14923.7495
EC00240=-0.7971,14927.5364
EC00241=-1.1939,14930.5396
EC00242=-0.5045,14932.2415
EC00243=-0.0057,14932.3197
EC00244=-0.0094,14932.2370
EC00245=-0.0188,14932.1156
EC00246=-0.0548,14932.0535
EC00247=8.4382,14932.8320
EC00248=26.6026,14935.8661
EC00249=28.1117,14938.3294
EC00250=28.1001,14940.0000
EC00251=28.1117,14941.6706
EC00252=26.6025,14944.1349
EC00253=8.4383,14947.1678
EC00254=-0.0548,14947.9465
EC00255=-0.0188,14947.8844
EC00256=-0.0094,14947.7630
EC00257=-0.0057,14947.6803
EC00258=-0.5045,14947.7585
EC00259=-1.1939,14949.4604
EC00260=-0.7971,14952.4636
EC00261=-0.0543,14956.2505
EC00262=-0.0054,14960.3860
EC00263=-0.0052,14964.6140
EC00264=-0.0540,14968.7498
EC00265=-0.7993,14972.5363
EC00266=-1.1940,14975.5394
EC00267=-0.5081,14977.2413
EC00268=-0.0087,14977.3191
EC00269=-0.0113,14977.2369
EC00270=-0.0208,14977.1159
EC00271=-0.0563,14977.0536
EC00272=8.4405,14977.8325
EC00273=26.5997,14980.8660
EC00274=28.1098,14983.3290
EC00275=28.0967,14985.0000
EC00276=28.1098,14986.6710
EC00277=26.5997,14989.1340
EC00278=8.4405,14992.1675
EC00279=-0.0563,14992.9464
EC00280=-0.0208,14992.8841
EC00281=-0.0113,14992.7631
EC00282=-0.0087,14992.6809
EC00283=-0.5081,14992.7587
EC00284=-1.1940,14994.4606
EC00285=-0.7993,14997.4637
EC00286=-0.0540,15001.2502
EC00287=-0.0052,15005.3860
EC00288=-0.0054,15009.6140
EC00289=-0.0543,15013.7495
EC00290=-0.7971,15017.5364
EC00291=-1.1939,15020.5396
EC00292=-0.5045,15022.2415
EC00293=-0.0057,15022.3197
EC00294=-0.0094,15022.2370
EC00295=-0.0188,15022.1156
EC00296=-0.0548,15022.0535
EC00297=8.4382,15022.8320
EC00298=26.6026,15025.8661
EC00299=28.1117,15028.3294
EC00300=28.1001,15030.0000
EC00301=28.1117,15031.6706
EC00302=26.6025,15034.1349
EC00303=8.4383,15037.1678
EC00304=-0.0548,15037.9465
EC00305=-0.0188,15037.8844
EC00306=-0.0094,15037.7630
EC00307=-0.0057,15037.6803
EC00308=-0.5045,15037.7585
EC00309=-1.1939,15039.4604
EC00310=-0.7971,15042.4636
EC00311=-0.0543,15046.2505
EC00312=-0.0054,15050.3860
EC00313=-0.0052,15054.6140
EC00314=-0.0540,15058.7498
EC00315=-0.7993,15062.5363
EC00316=-1.1940,15065.5394
EC00317=-0.5081,15067.2413
EC00318=-0.0087,15067.3191
EC00319=-0.0113,15067.2369
EC00320=-0.0208,15067.1159
EC00321=-0.0563,15067.0536
EC00322=8.4405,15067.8325
EC00323=26.5997,15070.8660
EC00324=28.1098,15073.3290
EC00325=28.0967,15075.0000
EC00326=28.1098,15076.6710
EC00327=26.5997,15079.1340
EC00328=8.4405,15082.1675
EC00329=-0.0563,15082.9464
EC00330=-0.0208,15082.8841
EC00331=-0.0113,15082.7631
EC00332=-0.0087,15082.6809
EC00333=-0.5081,15082.7587
EC00334=-1.1940,15084.4606
EC00335=-0.7993,15087.4637
EC00336=-0.0540,15091.2502
EC00337=-0.0052,15095.3860
EC00338=-0.0054,15099.6140
EC00339=-0.0543,15103.7495
EC00340=-0.7971,15107.5364
EC00341=-1.1939,15110.5396
EC00342=-0.5045,15112.2415
EC00343=-0.0057,15112.3197
EC00344=-0.0094,15112.2370
EC00345=-0.0188,15112.1156
EC00346=-0.0548,15112.0535
EC00347=8.4382,15112.8320
EC00348=26.6026,15115.8661
EC00349=28.1117,15118.3294
EC00350=28.1001,15120.0000
EC00351=28.1117,15121.6706
EC00352=26.6025,15124.1349
EC00353=8.4383,15127.1678
EC00354=-0.0548,15127.9465
EC00355=-0.0188,15127.8844
EC00356=-0.0094,15127.7630
EC00357=-0.0057,15127.6803
EC00358=-0.5045,15127.7585
EC00359=-1.1939,15129.4604
EC00360=-0.7971,15132.4636
EC00361=-0.0543,15136.2505
EC00362=-0.0054,15140.3860
EC00363=-0.0052,15144.6140
EC00364=-0.0540,15148.7498
EC00365=-0.7993,15152.5363
EC00366=-1.1940,15155.5394
EC00367=-0.5081,15157.2413
EC00368=-0.0087,15157.3191
EC00369=-0.0113,15157.2369
EC00370=-0.0208,15157.1159
EC00371=-0.0563,15157.0536
EC00372=8.4405,15157.8325
EC00373=26.5997,15160.8660
EC00374=28.1098,15163.3290
EC00375=28.0967,15165.0000
EC00376=28.1098,15166.6710
EC00377=26.5997,15169.1340
EC00378=8.4405,15172.1675
EC00379=-0.0563,15172.9464
EC00380=-0.0208,15172.8841
EC00381=-0.0113,15172.7631
EC00382=-0.0087,15172.6809
EC00383=-0.5081,15172.7587
EC00384=-1.1940,15174.4606
EC00385=-0.7993,15177.4637
EC00386=-0.0540,15181.2502
EC00387=-0.0052,15185.3860
EC00388=-0.0054,15189.6140
EC00389=-0.0543,15193.7495
EC00390=-0.7971,15197.5364
EC00391=-1.1939,15200.5396
EC00392=-0.5045,15202.2415
EC00393=-0.0057,15202.3197
EC00394=-0.0094,15202.2370
EC00395=-0.0188,15202.1156
EC00396=-0.0548,15202.0535
EC00397=8.4383,15202.8322
EC00398=26.6025,15205.8651
EC00399=28.1117,15208.3294
EC00400=26.2576,15210.0000
EC00401=26.2720,15211.6025
EC00402=24.7331,15214.0449
EC00403=7.3770,15217.0981
EC00404=-0.0435,15217.8538
EC00405=-0.0134,15217.7815
EC00406=-0.0020,15217.6711
EC00407=-0.0031,15217.6022
EC00408=-0.3615,15217.6844
EC00409=-0.8397,15219.3971
EC00410=-0.5442,15222.4165
EC00411=-0.0362,15226.2223
EC00412=-0.0054,15230.3773
EC00413=-0.0052,15234.6227
EC00414=-0.0384,15238.7775
EC00415=-0.5441,15242.5833
EC00416=-0.8412,15245.6027
EC00417=-0.3666,15247.3159
EC00418=-0.0016,15247.3980
EC00419=-0.0027,15247.3291
EC00420=-0.0129,15247.2193
EC00421=-0.0389,15247.1468
EC00422=7.3773,15247.9017
EC00423=24.7330,15250.9551
EC00424=26.2704,15253.3970
EC00425=26.2558,15255.0000
EC00426=26.2704,15256.6030
EC00427=24.7330,15259.0449
EC00428=7.3727,15262.0983
EC00429=-0.0389,15262.8532
EC00430=-0.0129,15262.7807
EC00431=-0.0027,15262.6709
EC00432=-0.0016,15262.6020
EC00433=-0.3666,15262.6841
EC00434=-0.8412,15264.3973
EC00435=-0.5441,15267.4167
EC00436=-0.0384,15271.2225
EC00437=-0.0052,15275.3773
EC00438=-0.0054,15279.6227
EC00439=-0.0362,15283.7777
EC00440=-0.5442,15287.5835
EC00441=-0.8397,15290.6029
EC00442=-0.3615,15292.3156
EC00443=-0.0031,15292.3978
EC00444=-0.0020,15292.3289
EC00445=-0.0134,15292.2185
EC00446=-0.0435,15292.1462
EC00447=7.3770,15292.9019
EC00448=24.7331,15295.9551
EC00449=26.2720,15298.3975
EC00450=26.2576,15300.0000
EC00451=26.2720,15301.6025
EC00452=24.7327,15304.0449
EC00453=7.3770,15307.0981
EC00454=-0.0435,15307.8538
EC00455=-0.0134,15307.7815
EC00456=-0.0020,15307.6711
EC00457=-0.0031,15307.6022
EC00458=-0.3615,15307.6844
EC00459=-0.8397,15309.3971
EC00460=-0.5442,15312.4165
EC00461=-0.0362,15316.2223
EC00462=-0.0054,15320.3773
EC00463=-0.0052,15324.6227
EC00464=-0.0384,15328.7775
EC00465=-0.5441,15332.5833
EC00466=-0.8412,15335.6027
EC00467=-0.3666,15337.3159
EC00468=-0.0016,15337.3980
EC00469=-0.0027,15337.3291
EC00470=-0.0129,15337.2193
EC00471=-0.0389,15337.1468
EC00472=7.3773,15337.9017
EC00473=24.7330,15340.9551
EC00474=26.2704,15343.3970
EC00475=26.2558,15345.0000
EC00476=26.2704,15346.6030
EC00477=24.7330,15349.0449
EC00478=7.3727,15352.0983
EC00479=-0.0389,15352.8532
EC00480=-0.0129,15352.7807
EC00481=-0.0027,15352.6709
EC00482=-0.0016,15352.6020
EC00483=-0.3666,15352.6841
EC00484=-0.8412,15354.3973
EC00485=-0.5441,15357.4167
EC00486=-0.0384,15361.2225
EC00487=-0.0052,15365.3773
EC00488=-0.0054,15369.6227
EC00489=-0.0362,15373.7777
EC00490=-0.5442,15377.5835
EC00491=-0.8397,15380.6029
EC00492=-0.3615,15382.3156
EC00493=-0.0031,15382.3978
EC00494=-0.0020,15382.3289
EC00495=-0.0134,15382.2185
EC00496=-0.0435,15382.1462
EC00497=7.3770,15382.9019
EC00498=24.7331,15385.9551
EC00499=26.2720,15388.3975
EC00500=26.2576,15390.0000
EC00501=26.2720,15391.6025
EC00502=24.7327,15394.0449
EC00503=7.3770,15397.0981
EC00504=-0.0435,15397.8538
EC00505=-0.0134,15397.7815
EC00506=-0.0020,15397.6711
EC00507=-0.0031,15397.6022
EC00508=-0.3615,15397.6844
EC00509=-0.8397,15399.3971
EC00510=-0.5442,15402.4165
EC00511=-0.0362,15406.2223
EC00512=-0.0054,15410.3773
EC00513=-0.0052,15414.6227
EC00514=-0.0384,15418.7775
EC00515=-0.5441,15422.5833
EC00516=-0.8412,15425.6027
EC00517=-0.3666,15427.3159
EC00518=-0.0016,15427.3980
EC00519=-0.0027,15427.3291
EC00520=-0.0129,15427.2193
EC00521=-0.0389,15427.1468
EC00522=7.3773,15427.9017
EC00523=24.7330,15430.9551
EC00524=26.2704,15433.3970
EC00525=26.2558,15435.0000
EC00526=26.2704,15436.6030
EC00527=24.7330,15439.0449
EC00528=7.3727,15442.0983
EC00529=-0.0389,15442.8532
EC00530=-0.0129,15442.7807
EC00531=-0.0027,15442.6709
EC00532=-0.0016,15442.6020
EC00533=-0.3666,15442.6841
EC00534=-0.8412,15444.3973
EC00535=-0.5441,15447.4167
EC00536=-0.0384,15451.2225
EC00537=-0.0052,15455.3773
EC00538=-0.0054,15459.6227
EC00539=-0.0362,15463.7777
EC00540=-0.5442,15467.5835
EC00541=-0.8397,15470.6029
EC00542=-0.3615,15472.3156
EC00543=-0.0031,15472.3978
EC00544=-0.0020,15472.3289
EC00545=-0.0134,15472.2185
EC00546=-0.0435,15472.1462
EC00547=7.3770,15472.9019
EC00548=24.7331,15475.9551
EC00549=26.2720,15478.3975
EC00550=26.2576,15480.0000
EC00551=26.2720,15481.6025
EC00552=24.7327,15484.0449
EC00553=7.3770,15487.0981
EC00554=-0.0435,15487.8538
EC00555=-0.0134,15487.7815
EC00556=-0.0020,15487.6711
EC00557=-0.0031,15487.6022
EC00558=-0.3615,15487.6844
EC00559=-0.8397,15489.3971
EC00560=-0.5442,15492.4165
EC00561=-0.0362,15496.2223
EC00562=-0.0054,15500.3773
EC00563=-0.0052,15504.6227
EC00564=-0.0384,15508.7775
EC00565=-0.5441,15512.5833
EC00566=-0.8412,15515.6027
EC00567=-0.3666,15517.3159
EC00568=-0.0016,15517.3980
EC00569=-0.0027,15517.3291
EC00570=-0.0129,15517.2193
EC00571=-0.0389,15517.1468
EC00572=7.3773,15517.9017
EC00573=24.7330,15520.9551
EC00574=26.2704,15523.3970
EC00575=26.2558,15525.0000
EC00576=26.2704,15526.6030
EC00577=24.7330,15529.0449
EC00578=7.3727,15532.0983
EC00579=-0.0389,15532.8532
EC00580=-0.0129,15532.7807
EC00581=-0.0027,15532.6709
EC00582=-0.0016,15532.6020
EC00583=-0.3666,15532.6841
EC00584=-0.8412,15534.3973
EC00585=-0.5441,15537.4167
EC00586=-0.0384,15541.2225
EC00587=-0.0052,15545.3773
EC00588=-0.0054,15549.6227
EC00589=-0.0362,15553.7777
EC00590=-0.5442,15557.5835
EC00591=-0.8397,15560.6029
EC00592=-0.3615,15562.3156
EC00593=-0.0031,15562.3978
EC00594=-0.0020,15562.3289
EC00595=-0.0134,15562.2185
EC00596=-0.0435,15562.1462
EC00597=7.3770,15562.9019
EC00598=24.7327,15565.9551
EC00599=26.2720,15568.3975
EC00600=24.1993,15570.0000
EC00601=24.2117,15571.5376
EC00602=22.6760,15573.9586
EC00603=6.3608,15577.0327
EC00604=-0.0296,15577.7683
EC00605=-0.0072,15577.6919
EC00606=0.0012,15577.5966
EC00607=0.0004,15577.5446
EC00608=-0.2180,15577.6343
EC00609=-0.4664,15579.3569
EC00610=-0.2743,15582.3884
EC00611=-0.0181,15586.2065
EC00612=-0.0000,15590.3718
EC00613=-0.0000,15594.6278
EC00614=-0.0128,15598.7938
EC00615=-0.2776,15602.6119
EC00616=-0.4673,15605.6434
EC00617=-0.2176,15607.3659
EC00618=0.0009,15607.4553
EC00619=-0.0015,15607.4027
EC00620=-0.0071,15607.3085
EC00621=-0.0275,15607.2322
EC00622=6.3616,15607.9674
EC00623=22.6775,15611.0417
EC00624=24.2122,15613.4634
EC00625=24.1961,15615.0000
EC00626=24.2160,15616.5366
EC00627=22.6769,15618.9583
EC00628=6.3616,15622.0326
EC00629=-0.0275,15622.7678
EC00630=-0.0071,15622.6915
EC00631=-0.0015,15622.5973
EC00632=0.0009,15622.5447
EC00633=-0.2176,15622.6341
EC00634=-0.4673,15624.3566
EC00635=-0.2776,15627.3881
EC00636=-0.0128,15631.2062
EC00637=-0.0000,15635.3722
EC00638=-0.0000,15639.6282
EC00639=-0.0181,15643.7935
EC00640=-0.2743,15647.6116
EC00641=-0.4664,15650.6431
EC00642=-0.2180,15652.3657
EC00643=0.0004,15652.4554
EC00644=0.0012,15652.4034
EC00645=-0.0072,15652.3081
EC00646=-0.0296,15652.2317
EC00647=6.3608,15652.9673
EC00648=22.6760,15656.0414
EC00649=24.2117,15658.4624
EC00650=24.1993,15660.0000
EC00651=24.2117,15661.5365
EC00652=22.6760,15663.9586
